(* Logix 5000 project; controller reports 1756-L63 rev 20.11; software revision 20.04; part 27 of 52 *)

        [1912].log_data[0].min := 1.0, [1912].log_data[0].max := 1.0, [1912].log_data[0].total := 300.0, [1912].log_data[0].time := 300.0, [1912].log_data[0].minminute := 40, [1912].log_data[0].maxminute := 40, [1912].log_data[0].valid := 1, [1912].log_data[1].valid := 1, [1912].log_data[2].valid := 1, [1912].log_data[3].valid := 1, [1912].log_data[4].valid := 1, [1912].log_data[5].valid := 1, [1912].log_data[6].valid := 1, [1912].log_data[7].valid := 1, [1912].log_data[8].valid := 1, [1912].log_data[9].valid := 1, [1912].log_data[10].valid := 1, [1912].log_data[11].valid := 1, [1912].log_data[12].valid := 1, [1912].log_data[13].valid := 1, [1912].log_data[14].valid := 1, [1912].log_data[15].valid := 1, [1912].log_data[16].valid := 1, [1912].log_data[17].valid := 1, [1912].log_data[18].valid := 1, [1912].log_data[19].valid := 1, [1912].time.Year := 2023, [1912].time.Month := 1, [1912].time.Day := 16, [1912].time.Hour := 7, [1912].time.Minute := 44, [1912].time.Second := 59, [1913].log_data[0].min := 1.0, [1913].log_data[0].max := 1.0, [1913].log_data[0].total := 300.0, [1913].log_data[0].time := 300.0, [1913].log_data[0].minminute := 45, [1913].log_data[0].maxminute := 45, [1913].log_data[0].valid := 1, [1913].log_data[1].valid := 1, [1913].log_data[2].valid := 1, [1913].log_data[3].valid := 1, [1913].log_data[4].valid := 1, [1913].log_data[5].valid := 1, [1913].log_data[6].valid := 1, [1913].log_data[7].valid := 1, [1913].log_data[8].valid := 1, [1913].log_data[9].valid := 1, [1913].log_data[10].valid := 1, [1913].log_data[11].valid := 1, [1913].log_data[12].valid := 1, [1913].log_data[13].valid := 1, [1913].log_data[14].valid := 1, [1913].log_data[15].valid := 1, [1913].log_data[16].valid := 1, [1913].log_data[17].valid := 1, [1913].log_data[18].valid := 1, [1913].log_data[19].valid := 1, [1913].time.Year := 2023, [1913].time.Month := 1,
        [1913].time.Day := 16, [1913].time.Hour := 7, [1913].time.Minute := 49, [1913].time.Second := 59, [1914].log_data[0].min := 1.0, [1914].log_data[0].max := 1.0, [1914].log_data[0].total := 300.0, [1914].log_data[0].time := 300.0, [1914].log_data[0].minminute := 50, [1914].log_data[0].maxminute := 50, [1914].log_data[0].valid := 1, [1914].log_data[1].valid := 1, [1914].log_data[2].valid := 1, [1914].log_data[3].valid := 1, [1914].log_data[4].valid := 1, [1914].log_data[5].valid := 1, [1914].log_data[6].valid := 1, [1914].log_data[7].valid := 1, [1914].log_data[8].valid := 1, [1914].log_data[9].valid := 1, [1914].log_data[10].valid := 1, [1914].log_data[11].valid := 1, [1914].log_data[12].valid := 1, [1914].log_data[13].valid := 1, [1914].log_data[14].valid := 1, [1914].log_data[15].valid := 1, [1914].log_data[16].valid := 1, [1914].log_data[17].valid := 1, [1914].log_data[18].valid := 1, [1914].log_data[19].valid := 1, [1914].time.Year := 2023, [1914].time.Month := 1, [1914].time.Day := 16, [1914].time.Hour := 7, [1914].time.Minute := 54, [1914].time.Second := 59, [1915].log_data[0].min := 1.0, [1915].log_data[0].max := 1.0, [1915].log_data[0].total := 300.0, [1915].log_data[0].time := 300.0, [1915].log_data[0].minminute := 55, [1915].log_data[0].maxminute := 55, [1915].log_data[0].valid := 1, [1915].log_data[1].valid := 1, [1915].log_data[2].valid := 1, [1915].log_data[3].valid := 1, [1915].log_data[4].valid := 1, [1915].log_data[5].valid := 1, [1915].log_data[6].valid := 1, [1915].log_data[7].valid := 1, [1915].log_data[8].valid := 1, [1915].log_data[9].valid := 1, [1915].log_data[10].valid := 1, [1915].log_data[11].valid := 1, [1915].log_data[12].valid := 1, [1915].log_data[13].valid := 1, [1915].log_data[14].valid := 1, [1915].log_data[15].valid := 1, [1915].log_data[16].valid := 1, [1915].log_data[17].valid := 1,
        [1915].log_data[18].valid := 1, [1915].log_data[19].valid := 1, [1915].time.Year := 2023, [1915].time.Month := 1, [1915].time.Day := 16, [1915].time.Hour := 7, [1915].time.Minute := 59, [1915].time.Second := 59, [1916].log_data[0].min := 1.0, [1916].log_data[0].max := 1.0, [1916].log_data[0].total := 300.0, [1916].log_data[0].time := 300.0, [1916].log_data[0].valid := 1, [1916].log_data[1].valid := 1, [1916].log_data[2].valid := 1, [1916].log_data[3].valid := 1, [1916].log_data[4].valid := 1, [1916].log_data[5].valid := 1, [1916].log_data[6].valid := 1, [1916].log_data[7].valid := 1, [1916].log_data[8].valid := 1, [1916].log_data[9].valid := 1, [1916].log_data[10].valid := 1, [1916].log_data[11].valid := 1, [1916].log_data[12].valid := 1, [1916].log_data[13].valid := 1, [1916].log_data[14].valid := 1, [1916].log_data[15].valid := 1, [1916].log_data[16].valid := 1, [1916].log_data[17].valid := 1, [1916].log_data[18].valid := 1, [1916].log_data[19].valid := 1, [1916].time.Year := 2023, [1916].time.Month := 1, [1916].time.Day := 16, [1916].time.Hour := 8, [1916].time.Minute := 4, [1916].time.Second := 59, [1917].log_data[0].min := 1.0, [1917].log_data[0].max := 1.0, [1917].log_data[0].total := 300.0, [1917].log_data[0].time := 300.0, [1917].log_data[0].minminute := 5, [1917].log_data[0].maxminute := 5, [1917].log_data[0].valid := 1, [1917].log_data[1].valid := 1, [1917].log_data[2].valid := 1, [1917].log_data[3].valid := 1, [1917].log_data[4].valid := 1, [1917].log_data[5].valid := 1, [1917].log_data[6].valid := 1, [1917].log_data[7].valid := 1, [1917].log_data[8].valid := 1, [1917].log_data[9].valid := 1, [1917].log_data[10].valid := 1, [1917].log_data[11].valid := 1, [1917].log_data[12].valid := 1, [1917].log_data[13].valid := 1, [1917].log_data[14].valid := 1, [1917].log_data[15].valid := 1,
        [1917].log_data[16].valid := 1, [1917].log_data[17].valid := 1, [1917].log_data[18].valid := 1, [1917].log_data[19].valid := 1, [1917].time.Year := 2023, [1917].time.Month := 1, [1917].time.Day := 16, [1917].time.Hour := 8, [1917].time.Minute := 9, [1917].time.Second := 59, [1918].log_data[0].min := 1.0, [1918].log_data[0].max := 1.0, [1918].log_data[0].total := 300.0, [1918].log_data[0].time := 300.0, [1918].log_data[0].minminute := 10, [1918].log_data[0].maxminute := 10, [1918].log_data[0].valid := 1, [1918].log_data[1].valid := 1, [1918].log_data[2].valid := 1, [1918].log_data[3].valid := 1, [1918].log_data[4].valid := 1, [1918].log_data[5].valid := 1, [1918].log_data[6].valid := 1, [1918].log_data[7].valid := 1, [1918].log_data[8].valid := 1, [1918].log_data[9].valid := 1, [1918].log_data[10].valid := 1, [1918].log_data[11].valid := 1, [1918].log_data[12].valid := 1, [1918].log_data[13].valid := 1, [1918].log_data[14].valid := 1, [1918].log_data[15].valid := 1, [1918].log_data[16].valid := 1, [1918].log_data[17].valid := 1, [1918].log_data[18].valid := 1, [1918].log_data[19].valid := 1, [1918].time.Year := 2023, [1918].time.Month := 1, [1918].time.Day := 16, [1918].time.Hour := 8, [1918].time.Minute := 14, [1918].time.Second := 59, [1919].log_data[0].min := 1.0, [1919].log_data[0].max := 1.0, [1919].log_data[0].total := 300.0, [1919].log_data[0].time := 300.0, [1919].log_data[0].minminute := 15, [1919].log_data[0].maxminute := 15, [1919].log_data[0].valid := 1, [1919].log_data[1].valid := 1, [1919].log_data[2].valid := 1, [1919].log_data[3].valid := 1, [1919].log_data[4].valid := 1, [1919].log_data[5].valid := 1, [1919].log_data[6].valid := 1, [1919].log_data[7].valid := 1, [1919].log_data[8].valid := 1, [1919].log_data[9].valid := 1, [1919].log_data[10].valid := 1, [1919].log_data[11].valid := 1,
        [1919].log_data[12].valid := 1, [1919].log_data[13].valid := 1, [1919].log_data[14].valid := 1, [1919].log_data[15].valid := 1, [1919].log_data[16].valid := 1, [1919].log_data[17].valid := 1, [1919].log_data[18].valid := 1, [1919].log_data[19].valid := 1, [1919].time.Year := 2023, [1919].time.Month := 1, [1919].time.Day := 16, [1919].time.Hour := 8, [1919].time.Minute := 19, [1919].time.Second := 59, [1920].log_data[0].min := 1.0, [1920].log_data[0].max := 1.0, [1920].log_data[0].total := 300.0, [1920].log_data[0].time := 300.0, [1920].log_data[0].minminute := 20, [1920].log_data[0].maxminute := 20, [1920].log_data[0].valid := 1, [1920].log_data[1].valid := 1, [1920].log_data[2].valid := 1, [1920].log_data[3].valid := 1, [1920].log_data[4].valid := 1, [1920].log_data[5].valid := 1, [1920].log_data[6].valid := 1, [1920].log_data[7].valid := 1, [1920].log_data[8].valid := 1, [1920].log_data[9].valid := 1, [1920].log_data[10].valid := 1, [1920].log_data[11].valid := 1, [1920].log_data[12].valid := 1, [1920].log_data[13].valid := 1, [1920].log_data[14].valid := 1, [1920].log_data[15].valid := 1, [1920].log_data[16].valid := 1, [1920].log_data[17].valid := 1, [1920].log_data[18].valid := 1, [1920].log_data[19].valid := 1, [1920].time.Year := 2023, [1920].time.Month := 1, [1920].time.Day := 16, [1920].time.Hour := 8, [1920].time.Minute := 24, [1920].time.Second := 59, [1921].log_data[0].min := 1.0, [1921].log_data[0].max := 1.0, [1921].log_data[0].total := 300.0, [1921].log_data[0].time := 300.0, [1921].log_data[0].minminute := 25, [1921].log_data[0].maxminute := 25, [1921].log_data[0].valid := 1, [1921].log_data[1].valid := 1, [1921].log_data[2].valid := 1, [1921].log_data[3].valid := 1, [1921].log_data[4].valid := 1, [1921].log_data[5].valid := 1, [1921].log_data[6].valid := 1, [1921].log_data[7].valid := 1,
        [1921].log_data[8].valid := 1, [1921].log_data[9].valid := 1, [1921].log_data[10].valid := 1, [1921].log_data[11].valid := 1, [1921].log_data[12].valid := 1, [1921].log_data[13].valid := 1, [1921].log_data[14].valid := 1, [1921].log_data[15].valid := 1, [1921].log_data[16].valid := 1, [1921].log_data[17].valid := 1, [1921].log_data[18].valid := 1, [1921].log_data[19].valid := 1, [1921].time.Year := 2023, [1921].time.Month := 1, [1921].time.Day := 16, [1921].time.Hour := 8, [1921].time.Minute := 29, [1921].time.Second := 59, [1922].log_data[0].min := 1.0, [1922].log_data[0].max := 1.0, [1922].log_data[0].total := 300.0, [1922].log_data[0].time := 300.0, [1922].log_data[0].minminute := 30, [1922].log_data[0].maxminute := 30, [1922].log_data[0].valid := 1, [1922].log_data[1].valid := 1, [1922].log_data[2].valid := 1, [1922].log_data[3].valid := 1, [1922].log_data[4].valid := 1, [1922].log_data[5].valid := 1, [1922].log_data[6].valid := 1, [1922].log_data[7].valid := 1, [1922].log_data[8].valid := 1, [1922].log_data[9].valid := 1, [1922].log_data[10].valid := 1, [1922].log_data[11].valid := 1, [1922].log_data[12].valid := 1, [1922].log_data[13].valid := 1, [1922].log_data[14].valid := 1, [1922].log_data[15].valid := 1, [1922].log_data[16].valid := 1, [1922].log_data[17].valid := 1, [1922].log_data[18].valid := 1, [1922].log_data[19].valid := 1, [1922].time.Year := 2023, [1922].time.Month := 1, [1922].time.Day := 16, [1922].time.Hour := 8, [1922].time.Minute := 34, [1922].time.Second := 59, [1923].log_data[0].min := 1.0, [1923].log_data[0].max := 1.0, [1923].log_data[0].total := 300.0, [1923].log_data[0].time := 300.0, [1923].log_data[0].minminute := 35, [1923].log_data[0].maxminute := 35, [1923].log_data[0].valid := 1, [1923].log_data[1].valid := 1, [1923].log_data[2].valid := 1, [1923].log_data[3].valid := 1,
        [1923].log_data[4].valid := 1, [1923].log_data[5].valid := 1, [1923].log_data[6].valid := 1, [1923].log_data[7].valid := 1, [1923].log_data[8].valid := 1, [1923].log_data[9].valid := 1, [1923].log_data[10].valid := 1, [1923].log_data[11].valid := 1, [1923].log_data[12].valid := 1, [1923].log_data[13].valid := 1, [1923].log_data[14].valid := 1, [1923].log_data[15].valid := 1, [1923].log_data[16].valid := 1, [1923].log_data[17].valid := 1, [1923].log_data[18].valid := 1, [1923].log_data[19].valid := 1, [1923].time.Year := 2023, [1923].time.Month := 1, [1923].time.Day := 16, [1923].time.Hour := 8, [1923].time.Minute := 39, [1923].time.Second := 59, [1924].log_data[0].min := 1.0, [1924].log_data[0].max := 1.0, [1924].log_data[0].total := 300.0, [1924].log_data[0].time := 300.0, [1924].log_data[0].minminute := 40, [1924].log_data[0].maxminute := 40, [1924].log_data[0].valid := 1, [1924].log_data[1].valid := 1, [1924].log_data[2].valid := 1, [1924].log_data[3].valid := 1, [1924].log_data[4].valid := 1, [1924].log_data[5].valid := 1, [1924].log_data[6].valid := 1, [1924].log_data[7].valid := 1, [1924].log_data[8].valid := 1, [1924].log_data[9].valid := 1, [1924].log_data[10].valid := 1, [1924].log_data[11].valid := 1, [1924].log_data[12].valid := 1, [1924].log_data[13].valid := 1, [1924].log_data[14].valid := 1, [1924].log_data[15].valid := 1, [1924].log_data[16].valid := 1, [1924].log_data[17].valid := 1, [1924].log_data[18].valid := 1, [1924].log_data[19].valid := 1, [1924].time.Year := 2023, [1924].time.Month := 1, [1924].time.Day := 16, [1924].time.Hour := 8, [1924].time.Minute := 44, [1924].time.Second := 59, [1925].log_data[0].min := 1.0, [1925].log_data[0].max := 1.0, [1925].log_data[0].total := 300.0, [1925].log_data[0].time := 300.0, [1925].log_data[0].minminute := 45, [1925].log_data[0].maxminute := 45,
        [1925].log_data[0].valid := 1, [1925].log_data[1].valid := 1, [1925].log_data[2].valid := 1, [1925].log_data[3].valid := 1, [1925].log_data[4].valid := 1, [1925].log_data[5].valid := 1, [1925].log_data[6].valid := 1, [1925].log_data[7].valid := 1, [1925].log_data[8].valid := 1, [1925].log_data[9].valid := 1, [1925].log_data[10].valid := 1, [1925].log_data[11].valid := 1, [1925].log_data[12].valid := 1, [1925].log_data[13].valid := 1, [1925].log_data[14].valid := 1, [1925].log_data[15].valid := 1, [1925].log_data[16].valid := 1, [1925].log_data[17].valid := 1, [1925].log_data[18].valid := 1, [1925].log_data[19].valid := 1, [1925].time.Year := 2023, [1925].time.Month := 1, [1925].time.Day := 16, [1925].time.Hour := 8, [1925].time.Minute := 49, [1925].time.Second := 59, [1926].log_data[0].min := 1.0, [1926].log_data[0].max := 1.0, [1926].log_data[0].total := 300.0, [1926].log_data[0].time := 300.0, [1926].log_data[0].minminute := 50, [1926].log_data[0].maxminute := 50, [1926].log_data[0].valid := 1, [1926].log_data[1].valid := 1, [1926].log_data[2].valid := 1, [1926].log_data[3].valid := 1, [1926].log_data[4].valid := 1, [1926].log_data[5].valid := 1, [1926].log_data[6].valid := 1, [1926].log_data[7].valid := 1, [1926].log_data[8].valid := 1, [1926].log_data[9].valid := 1, [1926].log_data[10].valid := 1, [1926].log_data[11].valid := 1, [1926].log_data[12].valid := 1, [1926].log_data[13].valid := 1, [1926].log_data[14].valid := 1, [1926].log_data[15].valid := 1, [1926].log_data[16].valid := 1, [1926].log_data[17].valid := 1, [1926].log_data[18].valid := 1, [1926].log_data[19].valid := 1, [1926].time.Year := 2023, [1926].time.Month := 1, [1926].time.Day := 16, [1926].time.Hour := 8, [1926].time.Minute := 54, [1926].time.Second := 59, [1927].log_data[0].min := 1.0, [1927].log_data[0].max := 1.0,
        [1927].log_data[0].total := 300.0, [1927].log_data[0].time := 300.0, [1927].log_data[0].minminute := 55, [1927].log_data[0].maxminute := 55, [1927].log_data[0].valid := 1, [1927].log_data[1].valid := 1, [1927].log_data[2].valid := 1, [1927].log_data[3].valid := 1, [1927].log_data[4].valid := 1, [1927].log_data[5].valid := 1, [1927].log_data[6].valid := 1, [1927].log_data[7].valid := 1, [1927].log_data[8].valid := 1, [1927].log_data[9].valid := 1, [1927].log_data[10].valid := 1, [1927].log_data[11].valid := 1, [1927].log_data[12].valid := 1, [1927].log_data[13].valid := 1, [1927].log_data[14].valid := 1, [1927].log_data[15].valid := 1, [1927].log_data[16].valid := 1, [1927].log_data[17].valid := 1, [1927].log_data[18].valid := 1, [1927].log_data[19].valid := 1, [1927].time.Year := 2023, [1927].time.Month := 1, [1927].time.Day := 16, [1927].time.Hour := 8, [1927].time.Minute := 59, [1927].time.Second := 59, [1928].log_data[0].min := 1.0, [1928].log_data[0].max := 1.0, [1928].log_data[0].total := 300.0, [1928].log_data[0].time := 300.0, [1928].log_data[0].valid := 1, [1928].log_data[1].valid := 1, [1928].log_data[2].valid := 1, [1928].log_data[3].valid := 1, [1928].log_data[4].valid := 1, [1928].log_data[5].valid := 1, [1928].log_data[6].valid := 1, [1928].log_data[7].valid := 1, [1928].log_data[8].valid := 1, [1928].log_data[9].valid := 1, [1928].log_data[10].valid := 1, [1928].log_data[11].valid := 1, [1928].log_data[12].valid := 1, [1928].log_data[13].valid := 1, [1928].log_data[14].valid := 1, [1928].log_data[15].valid := 1, [1928].log_data[16].valid := 1, [1928].log_data[17].valid := 1, [1928].log_data[18].valid := 1, [1928].log_data[19].valid := 1, [1928].time.Year := 2023, [1928].time.Month := 1, [1928].time.Day := 16, [1928].time.Hour := 9, [1928].time.Minute := 4, [1928].time.Second := 59,
        [1929].log_data[0].min := 1.0, [1929].log_data[0].max := 1.0, [1929].log_data[0].total := 300.0, [1929].log_data[0].time := 300.0, [1929].log_data[0].minminute := 5, [1929].log_data[0].maxminute := 5, [1929].log_data[0].valid := 1, [1929].log_data[1].valid := 1, [1929].log_data[2].valid := 1, [1929].log_data[3].valid := 1, [1929].log_data[4].valid := 1, [1929].log_data[5].valid := 1, [1929].log_data[6].valid := 1, [1929].log_data[7].valid := 1, [1929].log_data[8].valid := 1, [1929].log_data[9].valid := 1, [1929].log_data[10].valid := 1, [1929].log_data[11].valid := 1, [1929].log_data[12].valid := 1, [1929].log_data[13].valid := 1, [1929].log_data[14].valid := 1, [1929].log_data[15].valid := 1, [1929].log_data[16].valid := 1, [1929].log_data[17].valid := 1, [1929].log_data[18].valid := 1, [1929].log_data[19].valid := 1, [1929].time.Year := 2023, [1929].time.Month := 1, [1929].time.Day := 16, [1929].time.Hour := 9, [1929].time.Minute := 9, [1929].time.Second := 59, [1930].log_data[0].min := 1.0, [1930].log_data[0].max := 1.0, [1930].log_data[0].total := 300.0, [1930].log_data[0].time := 300.0, [1930].log_data[0].minminute := 10, [1930].log_data[0].maxminute := 10, [1930].log_data[0].valid := 1, [1930].log_data[1].valid := 1, [1930].log_data[2].valid := 1, [1930].log_data[3].valid := 1, [1930].log_data[4].valid := 1, [1930].log_data[5].valid := 1, [1930].log_data[6].valid := 1, [1930].log_data[7].valid := 1, [1930].log_data[8].valid := 1, [1930].log_data[9].valid := 1, [1930].log_data[10].valid := 1, [1930].log_data[11].valid := 1, [1930].log_data[12].valid := 1, [1930].log_data[13].valid := 1, [1930].log_data[14].valid := 1, [1930].log_data[15].valid := 1, [1930].log_data[16].valid := 1, [1930].log_data[17].valid := 1, [1930].log_data[18].valid := 1, [1930].log_data[19].valid := 1, [1930].time.Year := 2023, [1930].time.Month := 1,
        [1930].time.Day := 16, [1930].time.Hour := 9, [1930].time.Minute := 14, [1930].time.Second := 59, [1931].log_data[0].min := 1.0, [1931].log_data[0].max := 1.0, [1931].log_data[0].total := 300.0, [1931].log_data[0].time := 300.0, [1931].log_data[0].minminute := 15, [1931].log_data[0].maxminute := 15, [1931].log_data[0].valid := 1, [1931].log_data[1].valid := 1, [1931].log_data[2].valid := 1, [1931].log_data[3].valid := 1, [1931].log_data[4].valid := 1, [1931].log_data[5].valid := 1, [1931].log_data[6].valid := 1, [1931].log_data[7].valid := 1, [1931].log_data[8].valid := 1, [1931].log_data[9].valid := 1, [1931].log_data[10].valid := 1, [1931].log_data[11].valid := 1, [1931].log_data[12].valid := 1, [1931].log_data[13].valid := 1, [1931].log_data[14].valid := 1, [1931].log_data[15].valid := 1, [1931].log_data[16].valid := 1, [1931].log_data[17].valid := 1, [1931].log_data[18].valid := 1, [1931].log_data[19].valid := 1, [1931].time.Year := 2023, [1931].time.Month := 1, [1931].time.Day := 16, [1931].time.Hour := 9, [1931].time.Minute := 19, [1931].time.Second := 59, [1932].log_data[0].min := 1.0, [1932].log_data[0].max := 1.0, [1932].log_data[0].total := 300.0, [1932].log_data[0].time := 300.0, [1932].log_data[0].minminute := 20, [1932].log_data[0].maxminute := 20, [1932].log_data[0].valid := 1, [1932].log_data[1].valid := 1, [1932].log_data[2].valid := 1, [1932].log_data[3].valid := 1, [1932].log_data[4].valid := 1, [1932].log_data[5].valid := 1, [1932].log_data[6].valid := 1, [1932].log_data[7].valid := 1, [1932].log_data[8].valid := 1, [1932].log_data[9].valid := 1, [1932].log_data[10].valid := 1, [1932].log_data[11].valid := 1, [1932].log_data[12].valid := 1, [1932].log_data[13].valid := 1, [1932].log_data[14].valid := 1, [1932].log_data[15].valid := 1, [1932].log_data[16].valid := 1, [1932].log_data[17].valid := 1,
        [1932].log_data[18].valid := 1, [1932].log_data[19].valid := 1, [1932].time.Year := 2023, [1932].time.Month := 1, [1932].time.Day := 16, [1932].time.Hour := 9, [1932].time.Minute := 24, [1932].time.Second := 59, [1933].log_data[0].min := 1.0, [1933].log_data[0].max := 1.0, [1933].log_data[0].total := 300.0, [1933].log_data[0].time := 300.0, [1933].log_data[0].minminute := 25, [1933].log_data[0].maxminute := 25, [1933].log_data[0].valid := 1, [1933].log_data[1].valid := 1, [1933].log_data[2].valid := 1, [1933].log_data[3].valid := 1, [1933].log_data[4].valid := 1, [1933].log_data[5].valid := 1, [1933].log_data[6].valid := 1, [1933].log_data[7].valid := 1, [1933].log_data[8].valid := 1, [1933].log_data[9].valid := 1, [1933].log_data[10].valid := 1, [1933].log_data[11].valid := 1, [1933].log_data[12].valid := 1, [1933].log_data[13].valid := 1, [1933].log_data[14].valid := 1, [1933].log_data[15].valid := 1, [1933].log_data[16].valid := 1, [1933].log_data[17].valid := 1, [1933].log_data[18].valid := 1, [1933].log_data[19].valid := 1, [1933].time.Year := 2023, [1933].time.Month := 1, [1933].time.Day := 16, [1933].time.Hour := 9, [1933].time.Minute := 29, [1933].time.Second := 59, [1934].log_data[0].min := 1.0, [1934].log_data[0].max := 1.0, [1934].log_data[0].total := 300.0, [1934].log_data[0].time := 300.0, [1934].log_data[0].minminute := 30, [1934].log_data[0].maxminute := 30, [1934].log_data[0].valid := 1, [1934].log_data[1].valid := 1, [1934].log_data[2].valid := 1, [1934].log_data[3].valid := 1, [1934].log_data[4].valid := 1, [1934].log_data[5].valid := 1, [1934].log_data[6].valid := 1, [1934].log_data[7].valid := 1, [1934].log_data[8].valid := 1, [1934].log_data[9].valid := 1, [1934].log_data[10].valid := 1, [1934].log_data[11].valid := 1, [1934].log_data[12].valid := 1, [1934].log_data[13].valid := 1,
        [1934].log_data[14].valid := 1, [1934].log_data[15].valid := 1, [1934].log_data[16].valid := 1, [1934].log_data[17].valid := 1, [1934].log_data[18].valid := 1, [1934].log_data[19].valid := 1, [1934].time.Year := 2023, [1934].time.Month := 1, [1934].time.Day := 16, [1934].time.Hour := 9, [1934].time.Minute := 34, [1934].time.Second := 59, [1935].log_data[0].min := 1.0, [1935].log_data[0].max := 1.0, [1935].log_data[0].total := 300.0, [1935].log_data[0].time := 300.0, [1935].log_data[0].minminute := 35, [1935].log_data[0].maxminute := 35, [1935].log_data[0].valid := 1, [1935].log_data[1].valid := 1, [1935].log_data[2].valid := 1, [1935].log_data[3].valid := 1, [1935].log_data[4].valid := 1, [1935].log_data[5].valid := 1, [1935].log_data[6].valid := 1, [1935].log_data[7].valid := 1, [1935].log_data[8].valid := 1, [1935].log_data[9].valid := 1, [1935].log_data[10].valid := 1, [1935].log_data[11].valid := 1, [1935].log_data[12].valid := 1, [1935].log_data[13].valid := 1, [1935].log_data[14].valid := 1, [1935].log_data[15].valid := 1, [1935].log_data[16].valid := 1, [1935].log_data[17].valid := 1, [1935].log_data[18].valid := 1, [1935].log_data[19].valid := 1, [1935].time.Year := 2023, [1935].time.Month := 1, [1935].time.Day := 16, [1935].time.Hour := 9, [1935].time.Minute := 39, [1935].time.Second := 59, [1936].log_data[0].min := 1.0, [1936].log_data[0].max := 1.0, [1936].log_data[0].total := 300.0, [1936].log_data[0].time := 300.0, [1936].log_data[0].minminute := 40, [1936].log_data[0].maxminute := 40, [1936].log_data[0].valid := 1, [1936].log_data[1].valid := 1, [1936].log_data[2].valid := 1, [1936].log_data[3].valid := 1, [1936].log_data[4].valid := 1, [1936].log_data[5].valid := 1, [1936].log_data[6].valid := 1, [1936].log_data[7].valid := 1, [1936].log_data[8].valid := 1, [1936].log_data[9].valid := 1,
        [1936].log_data[10].valid := 1, [1936].log_data[11].valid := 1, [1936].log_data[12].valid := 1, [1936].log_data[13].valid := 1, [1936].log_data[14].valid := 1, [1936].log_data[15].valid := 1, [1936].log_data[16].valid := 1, [1936].log_data[17].valid := 1, [1936].log_data[18].valid := 1, [1936].log_data[19].valid := 1, [1936].time.Year := 2023, [1936].time.Month := 1, [1936].time.Day := 16, [1936].time.Hour := 9, [1936].time.Minute := 44, [1936].time.Second := 59, [1937].log_data[0].min := 1.0, [1937].log_data[0].max := 1.0, [1937].log_data[0].total := 300.0, [1937].log_data[0].time := 300.0, [1937].log_data[0].minminute := 45, [1937].log_data[0].maxminute := 45, [1937].log_data[0].valid := 1, [1937].log_data[1].valid := 1, [1937].log_data[2].valid := 1, [1937].log_data[3].valid := 1, [1937].log_data[4].valid := 1, [1937].log_data[5].valid := 1, [1937].log_data[6].valid := 1, [1937].log_data[7].valid := 1, [1937].log_data[8].valid := 1, [1937].log_data[9].valid := 1, [1937].log_data[10].valid := 1, [1937].log_data[11].valid := 1, [1937].log_data[12].valid := 1, [1937].log_data[13].valid := 1, [1937].log_data[14].valid := 1, [1937].log_data[15].valid := 1, [1937].log_data[16].valid := 1, [1937].log_data[17].valid := 1, [1937].log_data[18].valid := 1, [1937].log_data[19].valid := 1, [1937].time.Year := 2023, [1937].time.Month := 1, [1937].time.Day := 16, [1937].time.Hour := 9, [1937].time.Minute := 49, [1937].time.Second := 59, [1938].log_data[0].min := 1.0, [1938].log_data[0].max := 1.0, [1938].log_data[0].total := 300.0, [1938].log_data[0].time := 300.0, [1938].log_data[0].minminute := 50, [1938].log_data[0].maxminute := 50, [1938].log_data[0].valid := 1, [1938].log_data[1].valid := 1, [1938].log_data[2].valid := 1, [1938].log_data[3].valid := 1, [1938].log_data[4].valid := 1, [1938].log_data[5].valid := 1,
        [1938].log_data[6].valid := 1, [1938].log_data[7].valid := 1, [1938].log_data[8].valid := 1, [1938].log_data[9].valid := 1, [1938].log_data[10].valid := 1, [1938].log_data[11].valid := 1, [1938].log_data[12].valid := 1, [1938].log_data[13].valid := 1, [1938].log_data[14].valid := 1, [1938].log_data[15].valid := 1, [1938].log_data[16].valid := 1, [1938].log_data[17].valid := 1, [1938].log_data[18].valid := 1, [1938].log_data[19].valid := 1, [1938].time.Year := 2023, [1938].time.Month := 1, [1938].time.Day := 16, [1938].time.Hour := 9, [1938].time.Minute := 54, [1938].time.Second := 59, [1939].log_data[0].min := 1.0, [1939].log_data[0].max := 1.0, [1939].log_data[0].total := 300.0, [1939].log_data[0].time := 300.0, [1939].log_data[0].minminute := 55, [1939].log_data[0].maxminute := 55, [1939].log_data[0].valid := 1, [1939].log_data[1].valid := 1, [1939].log_data[2].valid := 1, [1939].log_data[3].valid := 1, [1939].log_data[4].valid := 1, [1939].log_data[5].valid := 1, [1939].log_data[6].valid := 1, [1939].log_data[7].valid := 1, [1939].log_data[8].valid := 1, [1939].log_data[9].valid := 1, [1939].log_data[10].valid := 1, [1939].log_data[11].valid := 1, [1939].log_data[12].valid := 1, [1939].log_data[13].valid := 1, [1939].log_data[14].valid := 1, [1939].log_data[15].valid := 1, [1939].log_data[16].valid := 1, [1939].log_data[17].valid := 1, [1939].log_data[18].valid := 1, [1939].log_data[19].valid := 1, [1939].time.Year := 2023, [1939].time.Month := 1, [1939].time.Day := 16, [1939].time.Hour := 9, [1939].time.Minute := 59, [1939].time.Second := 59, [1940].log_data[0].min := 1.0, [1940].log_data[0].max := 1.0, [1940].log_data[0].total := 299.5, [1940].log_data[0].time := 299.5, [1940].log_data[0].valid := 1, [1940].log_data[1].valid := 1, [1940].log_data[2].valid := 1, [1940].log_data[3].valid := 1,
        [1940].log_data[4].valid := 1, [1940].log_data[5].valid := 1, [1940].log_data[6].valid := 1, [1940].log_data[7].valid := 1, [1940].log_data[8].valid := 1, [1940].log_data[9].valid := 1, [1940].log_data[10].valid := 1, [1940].log_data[11].valid := 1, [1940].log_data[12].valid := 1, [1940].log_data[13].valid := 1, [1940].log_data[14].valid := 1, [1940].log_data[15].valid := 1, [1940].log_data[16].valid := 1, [1940].log_data[17].valid := 1, [1940].log_data[18].valid := 1, [1940].log_data[19].valid := 1, [1940].time.Year := 2023, [1940].time.Month := 1, [1940].time.Day := 16, [1940].time.Hour := 10, [1940].time.Minute := 4, [1940].time.Second := 59, [1941].log_data[0].min := 1.0, [1941].log_data[0].max := 1.0, [1941].log_data[0].total := 300.0, [1941].log_data[0].time := 300.0, [1941].log_data[0].minminute := 5, [1941].log_data[0].maxminute := 5, [1941].log_data[0].valid := 1, [1941].log_data[1].valid := 1, [1941].log_data[2].valid := 1, [1941].log_data[3].valid := 1, [1941].log_data[4].valid := 1, [1941].log_data[5].valid := 1, [1941].log_data[6].valid := 1, [1941].log_data[7].valid := 1, [1941].log_data[8].valid := 1, [1941].log_data[9].valid := 1, [1941].log_data[10].valid := 1, [1941].log_data[11].valid := 1, [1941].log_data[12].valid := 1, [1941].log_data[13].valid := 1, [1941].log_data[14].valid := 1, [1941].log_data[15].valid := 1, [1941].log_data[16].valid := 1, [1941].log_data[17].valid := 1, [1941].log_data[18].valid := 1, [1941].log_data[19].valid := 1, [1941].time.Year := 2023, [1941].time.Month := 1, [1941].time.Day := 16, [1941].time.Hour := 10, [1941].time.Minute := 9, [1941].time.Second := 59, [1942].log_data[0].min := 1.0, [1942].log_data[0].max := 1.0, [1942].log_data[0].total := 300.0, [1942].log_data[0].time := 300.0, [1942].log_data[0].minminute := 10, [1942].log_data[0].maxminute := 10,
        [1942].log_data[0].valid := 1, [1942].log_data[1].valid := 1, [1942].log_data[2].valid := 1, [1942].log_data[3].valid := 1, [1942].log_data[4].valid := 1, [1942].log_data[5].valid := 1, [1942].log_data[6].valid := 1, [1942].log_data[7].valid := 1, [1942].log_data[8].valid := 1, [1942].log_data[9].valid := 1, [1942].log_data[10].valid := 1, [1942].log_data[11].valid := 1, [1942].log_data[12].valid := 1, [1942].log_data[13].valid := 1, [1942].log_data[14].valid := 1, [1942].log_data[15].valid := 1, [1942].log_data[16].valid := 1, [1942].log_data[17].valid := 1, [1942].log_data[18].valid := 1, [1942].log_data[19].valid := 1, [1942].time.Year := 2023, [1942].time.Month := 1, [1942].time.Day := 16, [1942].time.Hour := 10, [1942].time.Minute := 14, [1942].time.Second := 59, [1943].log_data[0].min := 1.0, [1943].log_data[0].max := 1.0, [1943].log_data[0].total := 300.0, [1943].log_data[0].time := 300.0, [1943].log_data[0].minminute := 15, [1943].log_data[0].maxminute := 15, [1943].log_data[0].valid := 1, [1943].log_data[1].valid := 1, [1943].log_data[2].valid := 1, [1943].log_data[3].valid := 1, [1943].log_data[4].valid := 1, [1943].log_data[5].valid := 1, [1943].log_data[6].valid := 1, [1943].log_data[7].valid := 1, [1943].log_data[8].valid := 1, [1943].log_data[9].valid := 1, [1943].log_data[10].valid := 1, [1943].log_data[11].valid := 1, [1943].log_data[12].valid := 1, [1943].log_data[13].valid := 1, [1943].log_data[14].valid := 1, [1943].log_data[15].valid := 1, [1943].log_data[16].valid := 1, [1943].log_data[17].valid := 1, [1943].log_data[18].valid := 1, [1943].log_data[19].valid := 1, [1943].time.Year := 2023, [1943].time.Month := 1, [1943].time.Day := 16, [1943].time.Hour := 10, [1943].time.Minute := 19, [1943].time.Second := 59, [1944].log_data[0].min := 1.0, [1944].log_data[0].max := 1.0,
        [1944].log_data[0].total := 300.0, [1944].log_data[0].time := 300.0, [1944].log_data[0].minminute := 20, [1944].log_data[0].maxminute := 20, [1944].log_data[0].valid := 1, [1944].log_data[1].valid := 1, [1944].log_data[2].valid := 1, [1944].log_data[3].valid := 1, [1944].log_data[4].valid := 1, [1944].log_data[5].valid := 1, [1944].log_data[6].valid := 1, [1944].log_data[7].valid := 1, [1944].log_data[8].valid := 1, [1944].log_data[9].valid := 1, [1944].log_data[10].valid := 1, [1944].log_data[11].valid := 1, [1944].log_data[12].valid := 1, [1944].log_data[13].valid := 1, [1944].log_data[14].valid := 1, [1944].log_data[15].valid := 1, [1944].log_data[16].valid := 1, [1944].log_data[17].valid := 1, [1944].log_data[18].valid := 1, [1944].log_data[19].valid := 1, [1944].time.Year := 2023, [1944].time.Month := 1, [1944].time.Day := 16, [1944].time.Hour := 10, [1944].time.Minute := 24, [1944].time.Second := 59, [1945].log_data[0].min := 1.0, [1945].log_data[0].max := 1.0, [1945].log_data[0].total := 300.0, [1945].log_data[0].time := 300.0, [1945].log_data[0].minminute := 25, [1945].log_data[0].maxminute := 25, [1945].log_data[0].valid := 1, [1945].log_data[1].valid := 1, [1945].log_data[2].valid := 1, [1945].log_data[3].valid := 1, [1945].log_data[4].valid := 1, [1945].log_data[5].valid := 1, [1945].log_data[6].valid := 1, [1945].log_data[7].valid := 1, [1945].log_data[8].valid := 1, [1945].log_data[9].valid := 1, [1945].log_data[10].valid := 1, [1945].log_data[11].valid := 1, [1945].log_data[12].valid := 1, [1945].log_data[13].valid := 1, [1945].log_data[14].valid := 1, [1945].log_data[15].valid := 1, [1945].log_data[16].valid := 1, [1945].log_data[17].valid := 1, [1945].log_data[18].valid := 1, [1945].log_data[19].valid := 1, [1945].time.Year := 2023, [1945].time.Month := 1, [1945].time.Day := 16, [1945].time.Hour := 10,
        [1945].time.Minute := 29, [1945].time.Second := 59, [1946].log_data[0].min := 1.0, [1946].log_data[0].max := 1.0, [1946].log_data[0].total := 300.0, [1946].log_data[0].time := 300.0, [1946].log_data[0].minminute := 30, [1946].log_data[0].maxminute := 30, [1946].log_data[0].valid := 1, [1946].log_data[1].valid := 1, [1946].log_data[2].valid := 1, [1946].log_data[3].valid := 1, [1946].log_data[4].valid := 1, [1946].log_data[5].valid := 1, [1946].log_data[6].valid := 1, [1946].log_data[7].valid := 1, [1946].log_data[8].valid := 1, [1946].log_data[9].valid := 1, [1946].log_data[10].valid := 1, [1946].log_data[11].valid := 1, [1946].log_data[12].valid := 1, [1946].log_data[13].valid := 1, [1946].log_data[14].valid := 1, [1946].log_data[15].valid := 1, [1946].log_data[16].valid := 1, [1946].log_data[17].valid := 1, [1946].log_data[18].valid := 1, [1946].log_data[19].valid := 1, [1946].time.Year := 2023, [1946].time.Month := 1, [1946].time.Day := 16, [1946].time.Hour := 10, [1946].time.Minute := 34, [1946].time.Second := 59, [1947].log_data[0].min := 1.0, [1947].log_data[0].max := 1.0, [1947].log_data[0].total := 300.0, [1947].log_data[0].time := 300.0, [1947].log_data[0].minminute := 35, [1947].log_data[0].maxminute := 35, [1947].log_data[0].valid := 1, [1947].log_data[1].valid := 1, [1947].log_data[2].valid := 1, [1947].log_data[3].valid := 1, [1947].log_data[4].valid := 1, [1947].log_data[5].valid := 1, [1947].log_data[6].valid := 1, [1947].log_data[7].valid := 1, [1947].log_data[8].valid := 1, [1947].log_data[9].valid := 1, [1947].log_data[10].valid := 1, [1947].log_data[11].valid := 1, [1947].log_data[12].valid := 1, [1947].log_data[13].valid := 1, [1947].log_data[14].valid := 1, [1947].log_data[15].valid := 1, [1947].log_data[16].valid := 1, [1947].log_data[17].valid := 1, [1947].log_data[18].valid := 1, [1947].log_data[19].valid := 1,
        [1947].time.Year := 2023, [1947].time.Month := 1, [1947].time.Day := 16, [1947].time.Hour := 10, [1947].time.Minute := 39, [1947].time.Second := 59, [1948].log_data[0].min := 1.0, [1948].log_data[0].max := 1.0, [1948].log_data[0].total := 300.0, [1948].log_data[0].time := 300.0, [1948].log_data[0].minminute := 40, [1948].log_data[0].maxminute := 40, [1948].log_data[0].valid := 1, [1948].log_data[1].valid := 1, [1948].log_data[2].valid := 1, [1948].log_data[3].valid := 1, [1948].log_data[4].valid := 1, [1948].log_data[5].valid := 1, [1948].log_data[6].valid := 1, [1948].log_data[7].valid := 1, [1948].log_data[8].valid := 1, [1948].log_data[9].valid := 1, [1948].log_data[10].valid := 1, [1948].log_data[11].valid := 1, [1948].log_data[12].valid := 1, [1948].log_data[13].valid := 1, [1948].log_data[14].valid := 1, [1948].log_data[15].valid := 1, [1948].log_data[16].valid := 1, [1948].log_data[17].valid := 1, [1948].log_data[18].valid := 1, [1948].log_data[19].valid := 1, [1948].time.Year := 2023, [1948].time.Month := 1, [1948].time.Day := 16, [1948].time.Hour := 10, [1948].time.Minute := 44, [1948].time.Second := 59, [1949].log_data[0].min := 1.0, [1949].log_data[0].max := 1.0, [1949].log_data[0].total := 300.0, [1949].log_data[0].time := 300.0, [1949].log_data[0].minminute := 45, [1949].log_data[0].maxminute := 45, [1949].log_data[0].valid := 1, [1949].log_data[1].valid := 1, [1949].log_data[2].valid := 1, [1949].log_data[3].valid := 1, [1949].log_data[4].valid := 1, [1949].log_data[5].valid := 1, [1949].log_data[6].valid := 1, [1949].log_data[7].valid := 1, [1949].log_data[8].valid := 1, [1949].log_data[9].valid := 1, [1949].log_data[10].valid := 1, [1949].log_data[11].valid := 1, [1949].log_data[12].valid := 1, [1949].log_data[13].valid := 1, [1949].log_data[14].valid := 1, [1949].log_data[15].valid := 1,
        [1949].log_data[16].valid := 1, [1949].log_data[17].valid := 1, [1949].log_data[18].valid := 1, [1949].log_data[19].valid := 1, [1949].time.Year := 2023, [1949].time.Month := 1, [1949].time.Day := 16, [1949].time.Hour := 10, [1949].time.Minute := 49, [1949].time.Second := 59, [1950].log_data[0].min := 1.0, [1950].log_data[0].max := 1.0, [1950].log_data[0].total := 300.0, [1950].log_data[0].time := 300.0, [1950].log_data[0].minminute := 50, [1950].log_data[0].maxminute := 50, [1950].log_data[0].valid := 1, [1950].log_data[1].valid := 1, [1950].log_data[2].valid := 1, [1950].log_data[3].valid := 1, [1950].log_data[4].valid := 1, [1950].log_data[5].valid := 1, [1950].log_data[6].valid := 1, [1950].log_data[7].valid := 1, [1950].log_data[8].valid := 1, [1950].log_data[9].valid := 1, [1950].log_data[10].valid := 1, [1950].log_data[11].valid := 1, [1950].log_data[12].valid := 1, [1950].log_data[13].valid := 1, [1950].log_data[14].valid := 1, [1950].log_data[15].valid := 1, [1950].log_data[16].valid := 1, [1950].log_data[17].valid := 1, [1950].log_data[18].valid := 1, [1950].log_data[19].valid := 1, [1950].time.Year := 2023, [1950].time.Month := 1, [1950].time.Day := 16, [1950].time.Hour := 10, [1950].time.Minute := 54, [1950].time.Second := 59, [1951].log_data[0].min := 1.0, [1951].log_data[0].max := 1.0, [1951].log_data[0].total := 300.0, [1951].log_data[0].time := 300.0, [1951].log_data[0].minminute := 55, [1951].log_data[0].maxminute := 55, [1951].log_data[0].valid := 1, [1951].log_data[1].valid := 1, [1951].log_data[2].valid := 1, [1951].log_data[3].valid := 1, [1951].log_data[4].valid := 1, [1951].log_data[5].valid := 1, [1951].log_data[6].valid := 1, [1951].log_data[7].valid := 1, [1951].log_data[8].valid := 1, [1951].log_data[9].valid := 1, [1951].log_data[10].valid := 1, [1951].log_data[11].valid := 1,
        [1951].log_data[12].valid := 1, [1951].log_data[13].valid := 1, [1951].log_data[14].valid := 1, [1951].log_data[15].valid := 1, [1951].log_data[16].valid := 1, [1951].log_data[17].valid := 1, [1951].log_data[18].valid := 1, [1951].log_data[19].valid := 1, [1951].time.Year := 2023, [1951].time.Month := 1, [1951].time.Day := 16, [1951].time.Hour := 10, [1951].time.Minute := 59, [1951].time.Second := 59, [1952].log_data[0].min := 1.0, [1952].log_data[0].max := 1.0, [1952].log_data[0].total := 300.0, [1952].log_data[0].time := 300.0, [1952].log_data[0].valid := 1, [1952].log_data[1].valid := 1, [1952].log_data[2].valid := 1, [1952].log_data[3].valid := 1, [1952].log_data[4].valid := 1, [1952].log_data[5].valid := 1, [1952].log_data[6].valid := 1, [1952].log_data[7].valid := 1, [1952].log_data[8].valid := 1, [1952].log_data[9].valid := 1, [1952].log_data[10].valid := 1, [1952].log_data[11].valid := 1, [1952].log_data[12].valid := 1, [1952].log_data[13].valid := 1, [1952].log_data[14].valid := 1, [1952].log_data[15].valid := 1, [1952].log_data[16].valid := 1, [1952].log_data[17].valid := 1, [1952].log_data[18].valid := 1, [1952].log_data[19].valid := 1, [1952].time.Year := 2023, [1952].time.Month := 1, [1952].time.Day := 16, [1952].time.Hour := 11, [1952].time.Minute := 4, [1952].time.Second := 59, [1953].log_data[0].min := 1.0, [1953].log_data[0].max := 1.0, [1953].log_data[0].total := 300.0, [1953].log_data[0].time := 300.0, [1953].log_data[0].minminute := 5, [1953].log_data[0].maxminute := 5, [1953].log_data[0].valid := 1, [1953].log_data[1].valid := 1, [1953].log_data[2].valid := 1, [1953].log_data[3].valid := 1, [1953].log_data[4].valid := 1, [1953].log_data[5].valid := 1, [1953].log_data[6].valid := 1, [1953].log_data[7].valid := 1, [1953].log_data[8].valid := 1, [1953].log_data[9].valid := 1,
        [1953].log_data[10].valid := 1, [1953].log_data[11].valid := 1, [1953].log_data[12].valid := 1, [1953].log_data[13].valid := 1, [1953].log_data[14].valid := 1, [1953].log_data[15].valid := 1, [1953].log_data[16].valid := 1, [1953].log_data[17].valid := 1, [1953].log_data[18].valid := 1, [1953].log_data[19].valid := 1, [1953].time.Year := 2023, [1953].time.Month := 1, [1953].time.Day := 16, [1953].time.Hour := 11, [1953].time.Minute := 9, [1953].time.Second := 59, [1954].log_data[0].min := 1.0, [1954].log_data[0].max := 1.0, [1954].log_data[0].total := 300.0, [1954].log_data[0].time := 300.0, [1954].log_data[0].minminute := 10, [1954].log_data[0].maxminute := 10, [1954].log_data[0].valid := 1, [1954].log_data[1].valid := 1, [1954].log_data[2].valid := 1, [1954].log_data[3].valid := 1, [1954].log_data[4].valid := 1, [1954].log_data[5].valid := 1, [1954].log_data[6].valid := 1, [1954].log_data[7].valid := 1, [1954].log_data[8].valid := 1, [1954].log_data[9].valid := 1, [1954].log_data[10].valid := 1, [1954].log_data[11].valid := 1, [1954].log_data[12].valid := 1, [1954].log_data[13].valid := 1, [1954].log_data[14].valid := 1, [1954].log_data[15].valid := 1, [1954].log_data[16].valid := 1, [1954].log_data[17].valid := 1, [1954].log_data[18].valid := 1, [1954].log_data[19].valid := 1, [1954].time.Year := 2023, [1954].time.Month := 1, [1954].time.Day := 16, [1954].time.Hour := 11, [1954].time.Minute := 14, [1954].time.Second := 59, [1955].log_data[0].min := 1.0, [1955].log_data[0].max := 1.0, [1955].log_data[0].total := 300.0, [1955].log_data[0].time := 300.0, [1955].log_data[0].minminute := 15, [1955].log_data[0].maxminute := 15, [1955].log_data[0].valid := 1, [1955].log_data[1].valid := 1, [1955].log_data[2].valid := 1, [1955].log_data[3].valid := 1, [1955].log_data[4].valid := 1, [1955].log_data[5].valid := 1,
        [1955].log_data[6].valid := 1, [1955].log_data[7].valid := 1, [1955].log_data[8].valid := 1, [1955].log_data[9].valid := 1, [1955].log_data[10].valid := 1, [1955].log_data[11].valid := 1, [1955].log_data[12].valid := 1, [1955].log_data[13].valid := 1, [1955].log_data[14].valid := 1, [1955].log_data[15].valid := 1, [1955].log_data[16].valid := 1, [1955].log_data[17].valid := 1, [1955].log_data[18].valid := 1, [1955].log_data[19].valid := 1, [1955].time.Year := 2023, [1955].time.Month := 1, [1955].time.Day := 16, [1955].time.Hour := 11, [1955].time.Minute := 19, [1955].time.Second := 59, [1956].log_data[0].min := 1.0, [1956].log_data[0].max := 1.0, [1956].log_data[0].total := 300.0, [1956].log_data[0].time := 300.0, [1956].log_data[0].minminute := 20, [1956].log_data[0].maxminute := 20, [1956].log_data[0].valid := 1, [1956].log_data[1].valid := 1, [1956].log_data[2].valid := 1, [1956].log_data[3].valid := 1, [1956].log_data[4].valid := 1, [1956].log_data[5].valid := 1, [1956].log_data[6].valid := 1, [1956].log_data[7].valid := 1, [1956].log_data[8].valid := 1, [1956].log_data[9].valid := 1, [1956].log_data[10].valid := 1, [1956].log_data[11].valid := 1, [1956].log_data[12].valid := 1, [1956].log_data[13].valid := 1, [1956].log_data[14].valid := 1, [1956].log_data[15].valid := 1, [1956].log_data[16].valid := 1, [1956].log_data[17].valid := 1, [1956].log_data[18].valid := 1, [1956].log_data[19].valid := 1, [1956].time.Year := 2023, [1956].time.Month := 1, [1956].time.Day := 16, [1956].time.Hour := 11, [1956].time.Minute := 24, [1956].time.Second := 59, [1957].log_data[0].min := 1.0, [1957].log_data[0].max := 1.0, [1957].log_data[0].total := 300.0, [1957].log_data[0].time := 300.0, [1957].log_data[0].minminute := 25, [1957].log_data[0].maxminute := 25, [1957].log_data[0].valid := 1, [1957].log_data[1].valid := 1,
        [1957].log_data[2].valid := 1, [1957].log_data[3].valid := 1, [1957].log_data[4].valid := 1, [1957].log_data[5].valid := 1, [1957].log_data[6].valid := 1, [1957].log_data[7].valid := 1, [1957].log_data[8].valid := 1, [1957].log_data[9].valid := 1, [1957].log_data[10].valid := 1, [1957].log_data[11].valid := 1, [1957].log_data[12].valid := 1, [1957].log_data[13].valid := 1, [1957].log_data[14].valid := 1, [1957].log_data[15].valid := 1, [1957].log_data[16].valid := 1, [1957].log_data[17].valid := 1, [1957].log_data[18].valid := 1, [1957].log_data[19].valid := 1, [1957].time.Year := 2023, [1957].time.Month := 1, [1957].time.Day := 16, [1957].time.Hour := 11, [1957].time.Minute := 29, [1957].time.Second := 59, [1958].log_data[0].min := 1.0, [1958].log_data[0].max := 1.0, [1958].log_data[0].total := 300.0, [1958].log_data[0].time := 300.0, [1958].log_data[0].minminute := 30, [1958].log_data[0].maxminute := 30, [1958].log_data[0].valid := 1, [1958].log_data[1].valid := 1, [1958].log_data[2].valid := 1, [1958].log_data[3].valid := 1, [1958].log_data[4].valid := 1, [1958].log_data[5].valid := 1, [1958].log_data[6].valid := 1, [1958].log_data[7].valid := 1, [1958].log_data[8].valid := 1, [1958].log_data[9].valid := 1, [1958].log_data[10].valid := 1, [1958].log_data[11].valid := 1, [1958].log_data[12].valid := 1, [1958].log_data[13].valid := 1, [1958].log_data[14].valid := 1, [1958].log_data[15].valid := 1, [1958].log_data[16].valid := 1, [1958].log_data[17].valid := 1, [1958].log_data[18].valid := 1, [1958].log_data[19].valid := 1, [1958].time.Year := 2023, [1958].time.Month := 1, [1958].time.Day := 16, [1958].time.Hour := 11, [1958].time.Minute := 34, [1958].time.Second := 59, [1959].log_data[0].min := 1.0, [1959].log_data[0].max := 1.0, [1959].log_data[0].total := 300.0, [1959].log_data[0].time := 300.0,
        [1959].log_data[0].minminute := 35, [1959].log_data[0].maxminute := 35, [1959].log_data[0].valid := 1, [1959].log_data[1].valid := 1, [1959].log_data[2].valid := 1, [1959].log_data[3].valid := 1, [1959].log_data[4].valid := 1, [1959].log_data[5].valid := 1, [1959].log_data[6].valid := 1, [1959].log_data[7].valid := 1, [1959].log_data[8].valid := 1, [1959].log_data[9].valid := 1, [1959].log_data[10].valid := 1, [1959].log_data[11].valid := 1, [1959].log_data[12].valid := 1, [1959].log_data[13].valid := 1, [1959].log_data[14].valid := 1, [1959].log_data[15].valid := 1, [1959].log_data[16].valid := 1, [1959].log_data[17].valid := 1, [1959].log_data[18].valid := 1, [1959].log_data[19].valid := 1, [1959].time.Year := 2023, [1959].time.Month := 1, [1959].time.Day := 16, [1959].time.Hour := 11, [1959].time.Minute := 39, [1959].time.Second := 59, [1960].log_data[0].min := 1.0, [1960].log_data[0].max := 1.0, [1960].log_data[0].total := 300.0, [1960].log_data[0].time := 300.0, [1960].log_data[0].minminute := 40, [1960].log_data[0].maxminute := 40, [1960].log_data[0].valid := 1, [1960].log_data[1].valid := 1, [1960].log_data[2].valid := 1, [1960].log_data[3].valid := 1, [1960].log_data[4].valid := 1, [1960].log_data[5].valid := 1, [1960].log_data[6].valid := 1, [1960].log_data[7].valid := 1, [1960].log_data[8].valid := 1, [1960].log_data[9].valid := 1, [1960].log_data[10].valid := 1, [1960].log_data[11].valid := 1, [1960].log_data[12].valid := 1, [1960].log_data[13].valid := 1, [1960].log_data[14].valid := 1, [1960].log_data[15].valid := 1, [1960].log_data[16].valid := 1, [1960].log_data[17].valid := 1, [1960].log_data[18].valid := 1, [1960].log_data[19].valid := 1, [1960].time.Year := 2023, [1960].time.Month := 1, [1960].time.Day := 16, [1960].time.Hour := 11, [1960].time.Minute := 44, [1960].time.Second := 59,
        [1961].log_data[0].min := 1.0, [1961].log_data[0].max := 1.0, [1961].log_data[0].total := 300.0, [1961].log_data[0].time := 300.0, [1961].log_data[0].minminute := 45, [1961].log_data[0].maxminute := 45, [1961].log_data[0].valid := 1, [1961].log_data[1].valid := 1, [1961].log_data[2].valid := 1, [1961].log_data[3].valid := 1, [1961].log_data[4].valid := 1, [1961].log_data[5].valid := 1, [1961].log_data[6].valid := 1, [1961].log_data[7].valid := 1, [1961].log_data[8].valid := 1, [1961].log_data[9].valid := 1, [1961].log_data[10].valid := 1, [1961].log_data[11].valid := 1, [1961].log_data[12].valid := 1, [1961].log_data[13].valid := 1, [1961].log_data[14].valid := 1, [1961].log_data[15].valid := 1, [1961].log_data[16].valid := 1, [1961].log_data[17].valid := 1, [1961].log_data[18].valid := 1, [1961].log_data[19].valid := 1, [1961].time.Year := 2023, [1961].time.Month := 1, [1961].time.Day := 16, [1961].time.Hour := 11, [1961].time.Minute := 49, [1961].time.Second := 59, [1962].log_data[0].min := 1.0, [1962].log_data[0].max := 1.0, [1962].log_data[0].total := 300.0, [1962].log_data[0].time := 300.0, [1962].log_data[0].minminute := 50, [1962].log_data[0].maxminute := 50, [1962].log_data[0].valid := 1, [1962].log_data[1].valid := 1, [1962].log_data[2].valid := 1, [1962].log_data[3].valid := 1, [1962].log_data[4].valid := 1, [1962].log_data[5].valid := 1, [1962].log_data[6].valid := 1, [1962].log_data[7].valid := 1, [1962].log_data[8].valid := 1, [1962].log_data[9].valid := 1, [1962].log_data[10].valid := 1, [1962].log_data[11].valid := 1, [1962].log_data[12].valid := 1, [1962].log_data[13].valid := 1, [1962].log_data[14].valid := 1, [1962].log_data[15].valid := 1, [1962].log_data[16].valid := 1, [1962].log_data[17].valid := 1, [1962].log_data[18].valid := 1, [1962].log_data[19].valid := 1, [1962].time.Year := 2023, [1962].time.Month := 1,
        [1962].time.Day := 16, [1962].time.Hour := 11, [1962].time.Minute := 54, [1962].time.Second := 59, [1963].log_data[0].min := 1.0, [1963].log_data[0].max := 1.0, [1963].log_data[0].total := 300.0, [1963].log_data[0].time := 300.0, [1963].log_data[0].minminute := 55, [1963].log_data[0].maxminute := 55, [1963].log_data[0].valid := 1, [1963].log_data[1].valid := 1, [1963].log_data[2].valid := 1, [1963].log_data[3].valid := 1, [1963].log_data[4].valid := 1, [1963].log_data[5].valid := 1, [1963].log_data[6].valid := 1, [1963].log_data[7].valid := 1, [1963].log_data[8].valid := 1, [1963].log_data[9].valid := 1, [1963].log_data[10].valid := 1, [1963].log_data[11].valid := 1, [1963].log_data[12].valid := 1, [1963].log_data[13].valid := 1, [1963].log_data[14].valid := 1, [1963].log_data[15].valid := 1, [1963].log_data[16].valid := 1, [1963].log_data[17].valid := 1, [1963].log_data[18].valid := 1, [1963].log_data[19].valid := 1, [1963].time.Year := 2023, [1963].time.Month := 1, [1963].time.Day := 16, [1963].time.Hour := 11, [1963].time.Minute := 59, [1963].time.Second := 59, [1964].log_data[0].min := 1.0, [1964].log_data[0].max := 1.0, [1964].log_data[0].total := 300.0, [1964].log_data[0].time := 300.0, [1964].log_data[0].valid := 1, [1964].log_data[1].valid := 1, [1964].log_data[2].valid := 1, [1964].log_data[3].valid := 1, [1964].log_data[4].valid := 1, [1964].log_data[5].valid := 1, [1964].log_data[6].valid := 1, [1964].log_data[7].valid := 1, [1964].log_data[8].valid := 1, [1964].log_data[9].valid := 1, [1964].log_data[10].valid := 1, [1964].log_data[11].valid := 1, [1964].log_data[12].valid := 1, [1964].log_data[13].valid := 1, [1964].log_data[14].valid := 1, [1964].log_data[15].valid := 1, [1964].log_data[16].valid := 1, [1964].log_data[17].valid := 1, [1964].log_data[18].valid := 1, [1964].log_data[19].valid := 1,
        [1964].time.Year := 2023, [1964].time.Month := 1, [1964].time.Day := 16, [1964].time.Hour := 12, [1964].time.Minute := 4, [1964].time.Second := 59, [1965].log_data[0].min := 1.0, [1965].log_data[0].max := 1.0, [1965].log_data[0].total := 300.0, [1965].log_data[0].time := 300.0, [1965].log_data[0].minminute := 5, [1965].log_data[0].maxminute := 5, [1965].log_data[0].valid := 1, [1965].log_data[1].valid := 1, [1965].log_data[2].valid := 1, [1965].log_data[3].valid := 1, [1965].log_data[4].valid := 1, [1965].log_data[5].valid := 1, [1965].log_data[6].valid := 1, [1965].log_data[7].valid := 1, [1965].log_data[8].valid := 1, [1965].log_data[9].valid := 1, [1965].log_data[10].valid := 1, [1965].log_data[11].valid := 1, [1965].log_data[12].valid := 1, [1965].log_data[13].valid := 1, [1965].log_data[14].valid := 1, [1965].log_data[15].valid := 1, [1965].log_data[16].valid := 1, [1965].log_data[17].valid := 1, [1965].log_data[18].valid := 1, [1965].log_data[19].valid := 1, [1965].time.Year := 2023, [1965].time.Month := 1, [1965].time.Day := 16, [1965].time.Hour := 12, [1965].time.Minute := 9, [1965].time.Second := 59, [1966].log_data[0].min := 1.0, [1966].log_data[0].max := 1.0, [1966].log_data[0].total := 300.0, [1966].log_data[0].time := 300.0, [1966].log_data[0].minminute := 10, [1966].log_data[0].maxminute := 10, [1966].log_data[0].valid := 1, [1966].log_data[1].valid := 1, [1966].log_data[2].valid := 1, [1966].log_data[3].valid := 1, [1966].log_data[4].valid := 1, [1966].log_data[5].valid := 1, [1966].log_data[6].valid := 1, [1966].log_data[7].valid := 1, [1966].log_data[8].valid := 1, [1966].log_data[9].valid := 1, [1966].log_data[10].valid := 1, [1966].log_data[11].valid := 1, [1966].log_data[12].valid := 1, [1966].log_data[13].valid := 1, [1966].log_data[14].valid := 1, [1966].log_data[15].valid := 1,
        [1966].log_data[16].valid := 1, [1966].log_data[17].valid := 1, [1966].log_data[18].valid := 1, [1966].log_data[19].valid := 1, [1966].time.Year := 2023, [1966].time.Month := 1, [1966].time.Day := 16, [1966].time.Hour := 12, [1966].time.Minute := 14, [1966].time.Second := 59, [1967].log_data[0].min := 1.0, [1967].log_data[0].max := 1.0, [1967].log_data[0].total := 300.0, [1967].log_data[0].time := 300.0, [1967].log_data[0].minminute := 15, [1967].log_data[0].maxminute := 15, [1967].log_data[0].valid := 1, [1967].log_data[1].valid := 1, [1967].log_data[2].valid := 1, [1967].log_data[3].valid := 1, [1967].log_data[4].valid := 1, [1967].log_data[5].valid := 1, [1967].log_data[6].valid := 1, [1967].log_data[7].valid := 1, [1967].log_data[8].valid := 1, [1967].log_data[9].valid := 1, [1967].log_data[10].valid := 1, [1967].log_data[11].valid := 1, [1967].log_data[12].valid := 1, [1967].log_data[13].valid := 1, [1967].log_data[14].valid := 1, [1967].log_data[15].valid := 1, [1967].log_data[16].valid := 1, [1967].log_data[17].valid := 1, [1967].log_data[18].valid := 1, [1967].log_data[19].valid := 1, [1967].time.Year := 2023, [1967].time.Month := 1, [1967].time.Day := 16, [1967].time.Hour := 12, [1967].time.Minute := 19, [1967].time.Second := 59, [1968].log_data[0].min := 1.0, [1968].log_data[0].max := 1.0, [1968].log_data[0].total := 300.0, [1968].log_data[0].time := 300.0, [1968].log_data[0].minminute := 20, [1968].log_data[0].maxminute := 20, [1968].log_data[0].valid := 1, [1968].log_data[1].valid := 1, [1968].log_data[2].valid := 1, [1968].log_data[3].valid := 1, [1968].log_data[4].valid := 1, [1968].log_data[5].valid := 1, [1968].log_data[6].valid := 1, [1968].log_data[7].valid := 1, [1968].log_data[8].valid := 1, [1968].log_data[9].valid := 1, [1968].log_data[10].valid := 1, [1968].log_data[11].valid := 1,
        [1968].log_data[12].valid := 1, [1968].log_data[13].valid := 1, [1968].log_data[14].valid := 1, [1968].log_data[15].valid := 1, [1968].log_data[16].valid := 1, [1968].log_data[17].valid := 1, [1968].log_data[18].valid := 1, [1968].log_data[19].valid := 1, [1968].time.Year := 2023, [1968].time.Month := 1, [1968].time.Day := 16, [1968].time.Hour := 12, [1968].time.Minute := 24, [1968].time.Second := 59, [1969].log_data[0].min := 1.0, [1969].log_data[0].max := 1.0, [1969].log_data[0].total := 300.0, [1969].log_data[0].time := 300.0, [1969].log_data[0].minminute := 25, [1969].log_data[0].maxminute := 25, [1969].log_data[0].valid := 1, [1969].log_data[1].valid := 1, [1969].log_data[2].valid := 1, [1969].log_data[3].valid := 1, [1969].log_data[4].valid := 1, [1969].log_data[5].valid := 1, [1969].log_data[6].valid := 1, [1969].log_data[7].valid := 1, [1969].log_data[8].valid := 1, [1969].log_data[9].valid := 1, [1969].log_data[10].valid := 1, [1969].log_data[11].valid := 1, [1969].log_data[12].valid := 1, [1969].log_data[13].valid := 1, [1969].log_data[14].valid := 1, [1969].log_data[15].valid := 1, [1969].log_data[16].valid := 1, [1969].log_data[17].valid := 1, [1969].log_data[18].valid := 1, [1969].log_data[19].valid := 1, [1969].time.Year := 2023, [1969].time.Month := 1, [1969].time.Day := 16, [1969].time.Hour := 12, [1969].time.Minute := 29, [1969].time.Second := 59, [1970].log_data[0].min := 1.0, [1970].log_data[0].max := 1.0, [1970].log_data[0].total := 300.0, [1970].log_data[0].time := 300.0, [1970].log_data[0].minminute := 30, [1970].log_data[0].maxminute := 30, [1970].log_data[0].valid := 1, [1970].log_data[1].valid := 1, [1970].log_data[2].valid := 1, [1970].log_data[3].valid := 1, [1970].log_data[4].valid := 1, [1970].log_data[5].valid := 1, [1970].log_data[6].valid := 1, [1970].log_data[7].valid := 1,
        [1970].log_data[8].valid := 1, [1970].log_data[9].valid := 1, [1970].log_data[10].valid := 1, [1970].log_data[11].valid := 1, [1970].log_data[12].valid := 1, [1970].log_data[13].valid := 1, [1970].log_data[14].valid := 1, [1970].log_data[15].valid := 1, [1970].log_data[16].valid := 1, [1970].log_data[17].valid := 1, [1970].log_data[18].valid := 1, [1970].log_data[19].valid := 1, [1970].time.Year := 2023, [1970].time.Month := 1, [1970].time.Day := 16, [1970].time.Hour := 12, [1970].time.Minute := 34, [1970].time.Second := 59, [1971].log_data[0].min := 1.0, [1971].log_data[0].max := 1.0, [1971].log_data[0].total := 300.0, [1971].log_data[0].time := 300.0, [1971].log_data[0].minminute := 35, [1971].log_data[0].maxminute := 35, [1971].log_data[0].valid := 1, [1971].log_data[1].valid := 1, [1971].log_data[2].valid := 1, [1971].log_data[3].valid := 1, [1971].log_data[4].valid := 1, [1971].log_data[5].valid := 1, [1971].log_data[6].valid := 1, [1971].log_data[7].valid := 1, [1971].log_data[8].valid := 1, [1971].log_data[9].valid := 1, [1971].log_data[10].valid := 1, [1971].log_data[11].valid := 1, [1971].log_data[12].valid := 1, [1971].log_data[13].valid := 1, [1971].log_data[14].valid := 1, [1971].log_data[15].valid := 1, [1971].log_data[16].valid := 1, [1971].log_data[17].valid := 1, [1971].log_data[18].valid := 1, [1971].log_data[19].valid := 1, [1971].time.Year := 2023, [1971].time.Month := 1, [1971].time.Day := 16, [1971].time.Hour := 12, [1971].time.Minute := 39, [1971].time.Second := 59, [1972].log_data[0].min := 1.0, [1972].log_data[0].max := 1.0, [1972].log_data[0].total := 300.0, [1972].log_data[0].time := 300.0, [1972].log_data[0].minminute := 40, [1972].log_data[0].maxminute := 40, [1972].log_data[0].valid := 1, [1972].log_data[1].valid := 1, [1972].log_data[2].valid := 1, [1972].log_data[3].valid := 1,
        [1972].log_data[4].valid := 1, [1972].log_data[5].valid := 1, [1972].log_data[6].valid := 1, [1972].log_data[7].valid := 1, [1972].log_data[8].valid := 1, [1972].log_data[9].valid := 1, [1972].log_data[10].valid := 1, [1972].log_data[11].valid := 1, [1972].log_data[12].valid := 1, [1972].log_data[13].valid := 1, [1972].log_data[14].valid := 1, [1972].log_data[15].valid := 1, [1972].log_data[16].valid := 1, [1972].log_data[17].valid := 1, [1972].log_data[18].valid := 1, [1972].log_data[19].valid := 1, [1972].time.Year := 2023, [1972].time.Month := 1, [1972].time.Day := 16, [1972].time.Hour := 12, [1972].time.Minute := 44, [1972].time.Second := 59, [1973].log_data[0].min := 1.0, [1973].log_data[0].max := 1.0, [1973].log_data[0].total := 300.0, [1973].log_data[0].time := 300.0, [1973].log_data[0].minminute := 45, [1973].log_data[0].maxminute := 45, [1973].log_data[0].valid := 1, [1973].log_data[1].valid := 1, [1973].log_data[2].valid := 1, [1973].log_data[3].valid := 1, [1973].log_data[4].valid := 1, [1973].log_data[5].valid := 1, [1973].log_data[6].valid := 1, [1973].log_data[7].valid := 1, [1973].log_data[8].valid := 1, [1973].log_data[9].valid := 1, [1973].log_data[10].valid := 1, [1973].log_data[11].valid := 1, [1973].log_data[12].valid := 1, [1973].log_data[13].valid := 1, [1973].log_data[14].valid := 1, [1973].log_data[15].valid := 1, [1973].log_data[16].valid := 1, [1973].log_data[17].valid := 1, [1973].log_data[18].valid := 1, [1973].log_data[19].valid := 1, [1973].time.Year := 2023, [1973].time.Month := 1, [1973].time.Day := 16, [1973].time.Hour := 12, [1973].time.Minute := 49, [1973].time.Second := 59, [1974].log_data[0].min := 1.0, [1974].log_data[0].max := 1.0, [1974].log_data[0].total := 300.0, [1974].log_data[0].time := 300.0, [1974].log_data[0].minminute := 50, [1974].log_data[0].maxminute := 50,
        [1974].log_data[0].valid := 1, [1974].log_data[1].valid := 1, [1974].log_data[2].valid := 1, [1974].log_data[3].valid := 1, [1974].log_data[4].valid := 1, [1974].log_data[5].valid := 1, [1974].log_data[6].valid := 1, [1974].log_data[7].valid := 1, [1974].log_data[8].valid := 1, [1974].log_data[9].valid := 1, [1974].log_data[10].valid := 1, [1974].log_data[11].valid := 1, [1974].log_data[12].valid := 1, [1974].log_data[13].valid := 1, [1974].log_data[14].valid := 1, [1974].log_data[15].valid := 1, [1974].log_data[16].valid := 1, [1974].log_data[17].valid := 1, [1974].log_data[18].valid := 1, [1974].log_data[19].valid := 1, [1974].time.Year := 2023, [1974].time.Month := 1, [1974].time.Day := 16, [1974].time.Hour := 12, [1974].time.Minute := 54, [1974].time.Second := 59, [1975].log_data[0].min := 1.0, [1975].log_data[0].max := 1.0, [1975].log_data[0].total := 300.0, [1975].log_data[0].time := 300.0, [1975].log_data[0].minminute := 55, [1975].log_data[0].maxminute := 55, [1975].log_data[0].valid := 1, [1975].log_data[1].valid := 1, [1975].log_data[2].valid := 1, [1975].log_data[3].valid := 1, [1975].log_data[4].valid := 1, [1975].log_data[5].valid := 1, [1975].log_data[6].valid := 1, [1975].log_data[7].valid := 1, [1975].log_data[8].valid := 1, [1975].log_data[9].valid := 1, [1975].log_data[10].valid := 1, [1975].log_data[11].valid := 1, [1975].log_data[12].valid := 1, [1975].log_data[13].valid := 1, [1975].log_data[14].valid := 1, [1975].log_data[15].valid := 1, [1975].log_data[16].valid := 1, [1975].log_data[17].valid := 1, [1975].log_data[18].valid := 1, [1975].log_data[19].valid := 1, [1975].time.Year := 2023, [1975].time.Month := 1, [1975].time.Day := 16, [1975].time.Hour := 12, [1975].time.Minute := 59, [1975].time.Second := 59, [1976].log_data[0].min := 1.0, [1976].log_data[0].max := 1.0,
        [1976].log_data[0].total := 300.0, [1976].log_data[0].time := 300.0, [1976].log_data[0].valid := 1, [1976].log_data[1].valid := 1, [1976].log_data[2].valid := 1, [1976].log_data[3].valid := 1, [1976].log_data[4].valid := 1, [1976].log_data[5].valid := 1, [1976].log_data[6].valid := 1, [1976].log_data[7].valid := 1, [1976].log_data[8].valid := 1, [1976].log_data[9].valid := 1, [1976].log_data[10].valid := 1, [1976].log_data[11].valid := 1, [1976].log_data[12].valid := 1, [1976].log_data[13].valid := 1, [1976].log_data[14].valid := 1, [1976].log_data[15].valid := 1, [1976].log_data[16].valid := 1, [1976].log_data[17].valid := 1, [1976].log_data[18].valid := 1, [1976].log_data[19].valid := 1, [1976].time.Year := 2023, [1976].time.Month := 1, [1976].time.Day := 16, [1976].time.Hour := 13, [1976].time.Minute := 4, [1976].time.Second := 59, [1977].log_data[0].min := 1.0, [1977].log_data[0].max := 1.0, [1977].log_data[0].total := 300.0, [1977].log_data[0].time := 300.0, [1977].log_data[0].minminute := 5, [1977].log_data[0].maxminute := 5, [1977].log_data[0].valid := 1, [1977].log_data[1].valid := 1, [1977].log_data[2].valid := 1, [1977].log_data[3].valid := 1, [1977].log_data[4].valid := 1, [1977].log_data[5].valid := 1, [1977].log_data[6].valid := 1, [1977].log_data[7].valid := 1, [1977].log_data[8].valid := 1, [1977].log_data[9].valid := 1, [1977].log_data[10].valid := 1, [1977].log_data[11].valid := 1, [1977].log_data[12].valid := 1, [1977].log_data[13].valid := 1, [1977].log_data[14].valid := 1, [1977].log_data[15].valid := 1, [1977].log_data[16].valid := 1, [1977].log_data[17].valid := 1, [1977].log_data[18].valid := 1, [1977].log_data[19].valid := 1, [1977].time.Year := 2023, [1977].time.Month := 1, [1977].time.Day := 16, [1977].time.Hour := 13, [1977].time.Minute := 9, [1977].time.Second := 59,
        [1978].log_data[0].min := 1.0, [1978].log_data[0].max := 1.0, [1978].log_data[0].total := 300.0, [1978].log_data[0].time := 300.0, [1978].log_data[0].minminute := 10, [1978].log_data[0].maxminute := 10, [1978].log_data[0].valid := 1, [1978].log_data[1].valid := 1, [1978].log_data[2].valid := 1, [1978].log_data[3].valid := 1, [1978].log_data[4].valid := 1, [1978].log_data[5].valid := 1, [1978].log_data[6].valid := 1, [1978].log_data[7].valid := 1, [1978].log_data[8].valid := 1, [1978].log_data[9].valid := 1, [1978].log_data[10].valid := 1, [1978].log_data[11].valid := 1, [1978].log_data[12].valid := 1, [1978].log_data[13].valid := 1, [1978].log_data[14].valid := 1, [1978].log_data[15].valid := 1, [1978].log_data[16].valid := 1, [1978].log_data[17].valid := 1, [1978].log_data[18].valid := 1, [1978].log_data[19].valid := 1, [1978].time.Year := 2023, [1978].time.Month := 1, [1978].time.Day := 16, [1978].time.Hour := 13, [1978].time.Minute := 14, [1978].time.Second := 59, [1979].log_data[0].min := 1.0, [1979].log_data[0].max := 1.0, [1979].log_data[0].total := 300.0, [1979].log_data[0].time := 300.0, [1979].log_data[0].minminute := 15, [1979].log_data[0].maxminute := 15, [1979].log_data[0].valid := 1, [1979].log_data[1].valid := 1, [1979].log_data[2].valid := 1, [1979].log_data[3].valid := 1, [1979].log_data[4].valid := 1, [1979].log_data[5].valid := 1, [1979].log_data[6].valid := 1, [1979].log_data[7].valid := 1, [1979].log_data[8].valid := 1, [1979].log_data[9].valid := 1, [1979].log_data[10].valid := 1, [1979].log_data[11].valid := 1, [1979].log_data[12].valid := 1, [1979].log_data[13].valid := 1, [1979].log_data[14].valid := 1, [1979].log_data[15].valid := 1, [1979].log_data[16].valid := 1, [1979].log_data[17].valid := 1, [1979].log_data[18].valid := 1, [1979].log_data[19].valid := 1, [1979].time.Year := 2023, [1979].time.Month := 1,
        [1979].time.Day := 16, [1979].time.Hour := 13, [1979].time.Minute := 19, [1979].time.Second := 59, [1980].log_data[0].min := 1.0, [1980].log_data[0].max := 1.0, [1980].log_data[0].total := 300.0, [1980].log_data[0].time := 300.0, [1980].log_data[0].minminute := 20, [1980].log_data[0].maxminute := 20, [1980].log_data[0].valid := 1, [1980].log_data[1].valid := 1, [1980].log_data[2].valid := 1, [1980].log_data[3].valid := 1, [1980].log_data[4].valid := 1, [1980].log_data[5].valid := 1, [1980].log_data[6].valid := 1, [1980].log_data[7].valid := 1, [1980].log_data[8].valid := 1, [1980].log_data[9].valid := 1, [1980].log_data[10].valid := 1, [1980].log_data[11].valid := 1, [1980].log_data[12].valid := 1, [1980].log_data[13].valid := 1, [1980].log_data[14].valid := 1, [1980].log_data[15].valid := 1, [1980].log_data[16].valid := 1, [1980].log_data[17].valid := 1, [1980].log_data[18].valid := 1, [1980].log_data[19].valid := 1, [1980].time.Year := 2023, [1980].time.Month := 1, [1980].time.Day := 16, [1980].time.Hour := 13, [1980].time.Minute := 24, [1980].time.Second := 59, [1981].log_data[0].min := 1.0, [1981].log_data[0].max := 1.0, [1981].log_data[0].total := 300.0, [1981].log_data[0].time := 300.0, [1981].log_data[0].minminute := 25, [1981].log_data[0].maxminute := 25, [1981].log_data[0].valid := 1, [1981].log_data[1].valid := 1, [1981].log_data[2].valid := 1, [1981].log_data[3].valid := 1, [1981].log_data[4].valid := 1, [1981].log_data[5].valid := 1, [1981].log_data[6].valid := 1, [1981].log_data[7].valid := 1, [1981].log_data[8].valid := 1, [1981].log_data[9].valid := 1, [1981].log_data[10].valid := 1, [1981].log_data[11].valid := 1, [1981].log_data[12].valid := 1, [1981].log_data[13].valid := 1, [1981].log_data[14].valid := 1, [1981].log_data[15].valid := 1, [1981].log_data[16].valid := 1, [1981].log_data[17].valid := 1,
        [1981].log_data[18].valid := 1, [1981].log_data[19].valid := 1, [1981].time.Year := 2023, [1981].time.Month := 1, [1981].time.Day := 16, [1981].time.Hour := 13, [1981].time.Minute := 29, [1981].time.Second := 59, [1982].log_data[0].min := 1.0, [1982].log_data[0].max := 1.0, [1982].log_data[0].total := 300.0, [1982].log_data[0].time := 300.0, [1982].log_data[0].minminute := 30, [1982].log_data[0].maxminute := 30, [1982].log_data[0].valid := 1, [1982].log_data[1].valid := 1, [1982].log_data[2].valid := 1, [1982].log_data[3].valid := 1, [1982].log_data[4].valid := 1, [1982].log_data[5].valid := 1, [1982].log_data[6].valid := 1, [1982].log_data[7].valid := 1, [1982].log_data[8].valid := 1, [1982].log_data[9].valid := 1, [1982].log_data[10].valid := 1, [1982].log_data[11].valid := 1, [1982].log_data[12].valid := 1, [1982].log_data[13].valid := 1, [1982].log_data[14].valid := 1, [1982].log_data[15].valid := 1, [1982].log_data[16].valid := 1, [1982].log_data[17].valid := 1, [1982].log_data[18].valid := 1, [1982].log_data[19].valid := 1, [1982].time.Year := 2023, [1982].time.Month := 1, [1982].time.Day := 16, [1982].time.Hour := 13, [1982].time.Minute := 34, [1982].time.Second := 59, [1983].log_data[0].min := 1.0, [1983].log_data[0].max := 1.0, [1983].log_data[0].total := 300.0, [1983].log_data[0].time := 300.0, [1983].log_data[0].minminute := 35, [1983].log_data[0].maxminute := 35, [1983].log_data[0].valid := 1, [1983].log_data[1].valid := 1, [1983].log_data[2].valid := 1, [1983].log_data[3].valid := 1, [1983].log_data[4].valid := 1, [1983].log_data[5].valid := 1, [1983].log_data[6].valid := 1, [1983].log_data[7].valid := 1, [1983].log_data[8].valid := 1, [1983].log_data[9].valid := 1, [1983].log_data[10].valid := 1, [1983].log_data[11].valid := 1, [1983].log_data[12].valid := 1, [1983].log_data[13].valid := 1,
        [1983].log_data[14].valid := 1, [1983].log_data[15].valid := 1, [1983].log_data[16].valid := 1, [1983].log_data[17].valid := 1, [1983].log_data[18].valid := 1, [1983].log_data[19].valid := 1, [1983].time.Year := 2023, [1983].time.Month := 1, [1983].time.Day := 16, [1983].time.Hour := 13, [1983].time.Minute := 39, [1983].time.Second := 59, [1984].log_data[0].min := 1.0, [1984].log_data[0].max := 1.0, [1984].log_data[0].total := 300.0, [1984].log_data[0].time := 300.0, [1984].log_data[0].minminute := 40, [1984].log_data[0].maxminute := 40, [1984].log_data[0].valid := 1, [1984].log_data[1].valid := 1, [1984].log_data[2].valid := 1, [1984].log_data[3].valid := 1, [1984].log_data[4].valid := 1, [1984].log_data[5].valid := 1, [1984].log_data[6].valid := 1, [1984].log_data[7].valid := 1, [1984].log_data[8].valid := 1, [1984].log_data[9].valid := 1, [1984].log_data[10].valid := 1, [1984].log_data[11].valid := 1, [1984].log_data[12].valid := 1, [1984].log_data[13].valid := 1, [1984].log_data[14].valid := 1, [1984].log_data[15].valid := 1, [1984].log_data[16].valid := 1, [1984].log_data[17].valid := 1, [1984].log_data[18].valid := 1, [1984].log_data[19].valid := 1, [1984].time.Year := 2023, [1984].time.Month := 1, [1984].time.Day := 16, [1984].time.Hour := 13, [1984].time.Minute := 44, [1984].time.Second := 59, [1985].log_data[0].min := 1.0, [1985].log_data[0].max := 1.0, [1985].log_data[0].total := 300.0, [1985].log_data[0].time := 300.0, [1985].log_data[0].minminute := 45, [1985].log_data[0].maxminute := 45, [1985].log_data[0].valid := 1, [1985].log_data[1].valid := 1, [1985].log_data[2].valid := 1, [1985].log_data[3].valid := 1, [1985].log_data[4].valid := 1, [1985].log_data[5].valid := 1, [1985].log_data[6].valid := 1, [1985].log_data[7].valid := 1, [1985].log_data[8].valid := 1, [1985].log_data[9].valid := 1,
        [1985].log_data[10].valid := 1, [1985].log_data[11].valid := 1, [1985].log_data[12].valid := 1, [1985].log_data[13].valid := 1, [1985].log_data[14].valid := 1, [1985].log_data[15].valid := 1, [1985].log_data[16].valid := 1, [1985].log_data[17].valid := 1, [1985].log_data[18].valid := 1, [1985].log_data[19].valid := 1, [1985].time.Year := 2023, [1985].time.Month := 1, [1985].time.Day := 16, [1985].time.Hour := 13, [1985].time.Minute := 49, [1985].time.Second := 59, [1986].log_data[0].min := 1.0, [1986].log_data[0].max := 1.0, [1986].log_data[0].total := 300.0, [1986].log_data[0].time := 300.0, [1986].log_data[0].minminute := 50, [1986].log_data[0].maxminute := 50, [1986].log_data[0].valid := 1, [1986].log_data[1].valid := 1, [1986].log_data[2].valid := 1, [1986].log_data[3].valid := 1, [1986].log_data[4].valid := 1, [1986].log_data[5].valid := 1, [1986].log_data[6].valid := 1, [1986].log_data[7].valid := 1, [1986].log_data[8].valid := 1, [1986].log_data[9].valid := 1, [1986].log_data[10].valid := 1, [1986].log_data[11].valid := 1, [1986].log_data[12].valid := 1, [1986].log_data[13].valid := 1, [1986].log_data[14].valid := 1, [1986].log_data[15].valid := 1, [1986].log_data[16].valid := 1, [1986].log_data[17].valid := 1, [1986].log_data[18].valid := 1, [1986].log_data[19].valid := 1, [1986].time.Year := 2023, [1986].time.Month := 1, [1986].time.Day := 16, [1986].time.Hour := 13, [1986].time.Minute := 54, [1986].time.Second := 59, [1987].log_data[0].min := 1.0, [1987].log_data[0].max := 1.0, [1987].log_data[0].total := 300.0, [1987].log_data[0].time := 300.0, [1987].log_data[0].minminute := 55, [1987].log_data[0].maxminute := 55, [1987].log_data[0].valid := 1, [1987].log_data[1].valid := 1, [1987].log_data[2].valid := 1, [1987].log_data[3].valid := 1, [1987].log_data[4].valid := 1, [1987].log_data[5].valid := 1,
        [1987].log_data[6].valid := 1, [1987].log_data[7].valid := 1, [1987].log_data[8].valid := 1, [1987].log_data[9].valid := 1, [1987].log_data[10].valid := 1, [1987].log_data[11].valid := 1, [1987].log_data[12].valid := 1, [1987].log_data[13].valid := 1, [1987].log_data[14].valid := 1, [1987].log_data[15].valid := 1, [1987].log_data[16].valid := 1, [1987].log_data[17].valid := 1, [1987].log_data[18].valid := 1, [1987].log_data[19].valid := 1, [1987].time.Year := 2023, [1987].time.Month := 1, [1987].time.Day := 16, [1987].time.Hour := 13, [1987].time.Minute := 59, [1987].time.Second := 59, [1988].log_data[0].min := 1.0, [1988].log_data[0].max := 1.0, [1988].log_data[0].total := 300.0, [1988].log_data[0].time := 300.0, [1988].log_data[0].valid := 1, [1988].log_data[1].valid := 1, [1988].log_data[2].valid := 1, [1988].log_data[3].valid := 1, [1988].log_data[4].valid := 1, [1988].log_data[5].valid := 1, [1988].log_data[6].valid := 1, [1988].log_data[7].valid := 1, [1988].log_data[8].valid := 1, [1988].log_data[9].valid := 1, [1988].log_data[10].valid := 1, [1988].log_data[11].valid := 1, [1988].log_data[12].valid := 1, [1988].log_data[13].valid := 1, [1988].log_data[14].valid := 1, [1988].log_data[15].valid := 1, [1988].log_data[16].valid := 1, [1988].log_data[17].valid := 1, [1988].log_data[18].valid := 1, [1988].log_data[19].valid := 1, [1988].time.Year := 2023, [1988].time.Month := 1, [1988].time.Day := 16, [1988].time.Hour := 14, [1988].time.Minute := 4, [1988].time.Second := 59, [1989].log_data[0].min := 1.0, [1989].log_data[0].max := 1.0, [1989].log_data[0].total := 300.0, [1989].log_data[0].time := 300.0, [1989].log_data[0].minminute := 5, [1989].log_data[0].maxminute := 5, [1989].log_data[0].valid := 1, [1989].log_data[1].valid := 1, [1989].log_data[2].valid := 1, [1989].log_data[3].valid := 1,
        [1989].log_data[4].valid := 1, [1989].log_data[5].valid := 1, [1989].log_data[6].valid := 1, [1989].log_data[7].valid := 1, [1989].log_data[8].valid := 1, [1989].log_data[9].valid := 1, [1989].log_data[10].valid := 1, [1989].log_data[11].valid := 1, [1989].log_data[12].valid := 1, [1989].log_data[13].valid := 1, [1989].log_data[14].valid := 1, [1989].log_data[15].valid := 1, [1989].log_data[16].valid := 1, [1989].log_data[17].valid := 1, [1989].log_data[18].valid := 1, [1989].log_data[19].valid := 1, [1989].time.Year := 2023, [1989].time.Month := 1, [1989].time.Day := 16, [1989].time.Hour := 14, [1989].time.Minute := 9, [1989].time.Second := 59, [1990].log_data[0].min := 1.0, [1990].log_data[0].max := 1.0, [1990].log_data[0].total := 300.0, [1990].log_data[0].time := 300.0, [1990].log_data[0].minminute := 10, [1990].log_data[0].maxminute := 10, [1990].log_data[0].valid := 1, [1990].log_data[1].valid := 1, [1990].log_data[2].valid := 1, [1990].log_data[3].valid := 1, [1990].log_data[4].valid := 1, [1990].log_data[5].valid := 1, [1990].log_data[6].valid := 1, [1990].log_data[7].valid := 1, [1990].log_data[8].valid := 1, [1990].log_data[9].valid := 1, [1990].log_data[10].valid := 1, [1990].log_data[11].valid := 1, [1990].log_data[12].valid := 1, [1990].log_data[13].valid := 1, [1990].log_data[14].valid := 1, [1990].log_data[15].valid := 1, [1990].log_data[16].valid := 1, [1990].log_data[17].valid := 1, [1990].log_data[18].valid := 1, [1990].log_data[19].valid := 1, [1990].time.Year := 2023, [1990].time.Month := 1, [1990].time.Day := 16, [1990].time.Hour := 14, [1990].time.Minute := 14, [1990].time.Second := 59, [1991].log_data[0].min := 1.0, [1991].log_data[0].max := 1.0, [1991].log_data[0].total := 300.0, [1991].log_data[0].time := 300.0, [1991].log_data[0].minminute := 15, [1991].log_data[0].maxminute := 15,
        [1991].log_data[0].valid := 1, [1991].log_data[1].valid := 1, [1991].log_data[2].valid := 1, [1991].log_data[3].valid := 1, [1991].log_data[4].valid := 1, [1991].log_data[5].valid := 1, [1991].log_data[6].valid := 1, [1991].log_data[7].valid := 1, [1991].log_data[8].valid := 1, [1991].log_data[9].valid := 1, [1991].log_data[10].valid := 1, [1991].log_data[11].valid := 1, [1991].log_data[12].valid := 1, [1991].log_data[13].valid := 1, [1991].log_data[14].valid := 1, [1991].log_data[15].valid := 1, [1991].log_data[16].valid := 1, [1991].log_data[17].valid := 1, [1991].log_data[18].valid := 1, [1991].log_data[19].valid := 1, [1991].time.Year := 2023, [1991].time.Month := 1, [1991].time.Day := 16, [1991].time.Hour := 14, [1991].time.Minute := 19, [1991].time.Second := 59, [1992].log_data[0].min := 1.0, [1992].log_data[0].max := 1.0, [1992].log_data[0].total := 300.0, [1992].log_data[0].time := 300.0, [1992].log_data[0].minminute := 20, [1992].log_data[0].maxminute := 20, [1992].log_data[0].valid := 1, [1992].log_data[1].valid := 1, [1992].log_data[2].valid := 1, [1992].log_data[3].valid := 1, [1992].log_data[4].valid := 1, [1992].log_data[5].valid := 1, [1992].log_data[6].valid := 1, [1992].log_data[7].valid := 1, [1992].log_data[8].valid := 1, [1992].log_data[9].valid := 1, [1992].log_data[10].valid := 1, [1992].log_data[11].valid := 1, [1992].log_data[12].valid := 1, [1992].log_data[13].valid := 1, [1992].log_data[14].valid := 1, [1992].log_data[15].valid := 1, [1992].log_data[16].valid := 1, [1992].log_data[17].valid := 1, [1992].log_data[18].valid := 1, [1992].log_data[19].valid := 1, [1992].time.Year := 2023, [1992].time.Month := 1, [1992].time.Day := 16, [1992].time.Hour := 14, [1992].time.Minute := 24, [1992].time.Second := 59, [1993].log_data[0].min := 1.0, [1993].log_data[0].max := 1.0,
        [1993].log_data[0].total := 300.0, [1993].log_data[0].time := 300.0, [1993].log_data[0].minminute := 25, [1993].log_data[0].maxminute := 25, [1993].log_data[0].valid := 1, [1993].log_data[1].valid := 1, [1993].log_data[2].valid := 1, [1993].log_data[3].valid := 1, [1993].log_data[4].valid := 1, [1993].log_data[5].valid := 1, [1993].log_data[6].valid := 1, [1993].log_data[7].valid := 1, [1993].log_data[8].valid := 1, [1993].log_data[9].valid := 1, [1993].log_data[10].valid := 1, [1993].log_data[11].valid := 1, [1993].log_data[12].valid := 1, [1993].log_data[13].valid := 1, [1993].log_data[14].valid := 1, [1993].log_data[15].valid := 1, [1993].log_data[16].valid := 1, [1993].log_data[17].valid := 1, [1993].log_data[18].valid := 1, [1993].log_data[19].valid := 1, [1993].time.Year := 2023, [1993].time.Month := 1, [1993].time.Day := 16, [1993].time.Hour := 14, [1993].time.Minute := 29, [1993].time.Second := 59, [1994].log_data[0].min := 1.0, [1994].log_data[0].max := 1.0, [1994].log_data[0].total := 300.0, [1994].log_data[0].time := 300.0, [1994].log_data[0].minminute := 30, [1994].log_data[0].maxminute := 30, [1994].log_data[0].valid := 1, [1994].log_data[1].valid := 1, [1994].log_data[2].valid := 1, [1994].log_data[3].valid := 1, [1994].log_data[4].valid := 1, [1994].log_data[5].valid := 1, [1994].log_data[6].valid := 1, [1994].log_data[7].valid := 1, [1994].log_data[8].valid := 1, [1994].log_data[9].valid := 1, [1994].log_data[10].valid := 1, [1994].log_data[11].valid := 1, [1994].log_data[12].valid := 1, [1994].log_data[13].valid := 1, [1994].log_data[14].valid := 1, [1994].log_data[15].valid := 1, [1994].log_data[16].valid := 1, [1994].log_data[17].valid := 1, [1994].log_data[18].valid := 1, [1994].log_data[19].valid := 1, [1994].time.Year := 2023, [1994].time.Month := 1, [1994].time.Day := 16, [1994].time.Hour := 14,
        [1994].time.Minute := 34, [1994].time.Second := 59, [1995].log_data[0].min := 1.0, [1995].log_data[0].max := 1.0, [1995].log_data[0].total := 300.0, [1995].log_data[0].time := 300.0, [1995].log_data[0].minminute := 35, [1995].log_data[0].maxminute := 35, [1995].log_data[0].valid := 1, [1995].log_data[1].valid := 1, [1995].log_data[2].valid := 1, [1995].log_data[3].valid := 1, [1995].log_data[4].valid := 1, [1995].log_data[5].valid := 1, [1995].log_data[6].valid := 1, [1995].log_data[7].valid := 1, [1995].log_data[8].valid := 1, [1995].log_data[9].valid := 1, [1995].log_data[10].valid := 1, [1995].log_data[11].valid := 1, [1995].log_data[12].valid := 1, [1995].log_data[13].valid := 1, [1995].log_data[14].valid := 1, [1995].log_data[15].valid := 1, [1995].log_data[16].valid := 1, [1995].log_data[17].valid := 1, [1995].log_data[18].valid := 1, [1995].log_data[19].valid := 1, [1995].time.Year := 2023, [1995].time.Month := 1, [1995].time.Day := 16, [1995].time.Hour := 14, [1995].time.Minute := 39, [1995].time.Second := 59, [1996].log_data[0].min := 1.0, [1996].log_data[0].max := 1.0, [1996].log_data[0].total := 300.0, [1996].log_data[0].time := 300.0, [1996].log_data[0].minminute := 40, [1996].log_data[0].maxminute := 40, [1996].log_data[0].valid := 1, [1996].log_data[1].valid := 1, [1996].log_data[2].valid := 1, [1996].log_data[3].valid := 1, [1996].log_data[4].valid := 1, [1996].log_data[5].valid := 1, [1996].log_data[6].valid := 1, [1996].log_data[7].valid := 1, [1996].log_data[8].valid := 1, [1996].log_data[9].valid := 1, [1996].log_data[10].valid := 1, [1996].log_data[11].valid := 1, [1996].log_data[12].valid := 1, [1996].log_data[13].valid := 1, [1996].log_data[14].valid := 1, [1996].log_data[15].valid := 1, [1996].log_data[16].valid := 1, [1996].log_data[17].valid := 1, [1996].log_data[18].valid := 1, [1996].log_data[19].valid := 1,
        [1996].time.Year := 2023, [1996].time.Month := 1, [1996].time.Day := 16, [1996].time.Hour := 14, [1996].time.Minute := 44, [1996].time.Second := 59, [1997].log_data[0].min := 1.0, [1997].log_data[0].max := 1.0, [1997].log_data[0].total := 300.0, [1997].log_data[0].time := 300.0, [1997].log_data[0].minminute := 45, [1997].log_data[0].maxminute := 45, [1997].log_data[0].valid := 1, [1997].log_data[1].valid := 1, [1997].log_data[2].valid := 1, [1997].log_data[3].valid := 1, [1997].log_data[4].valid := 1, [1997].log_data[5].valid := 1, [1997].log_data[6].valid := 1, [1997].log_data[7].valid := 1, [1997].log_data[8].valid := 1, [1997].log_data[9].valid := 1, [1997].log_data[10].valid := 1, [1997].log_data[11].valid := 1, [1997].log_data[12].valid := 1, [1997].log_data[13].valid := 1, [1997].log_data[14].valid := 1, [1997].log_data[15].valid := 1, [1997].log_data[16].valid := 1, [1997].log_data[17].valid := 1, [1997].log_data[18].valid := 1, [1997].log_data[19].valid := 1, [1997].time.Year := 2023, [1997].time.Month := 1, [1997].time.Day := 16, [1997].time.Hour := 14, [1997].time.Minute := 49, [1997].time.Second := 59, [1998].log_data[0].min := 1.0, [1998].log_data[0].max := 1.0, [1998].log_data[0].total := 300.0, [1998].log_data[0].time := 300.0, [1998].log_data[0].minminute := 50, [1998].log_data[0].maxminute := 50, [1998].log_data[0].valid := 1, [1998].log_data[1].valid := 1, [1998].log_data[2].valid := 1, [1998].log_data[3].valid := 1, [1998].log_data[4].valid := 1, [1998].log_data[5].valid := 1, [1998].log_data[6].valid := 1, [1998].log_data[7].valid := 1, [1998].log_data[8].valid := 1, [1998].log_data[9].valid := 1, [1998].log_data[10].valid := 1, [1998].log_data[11].valid := 1, [1998].log_data[12].valid := 1, [1998].log_data[13].valid := 1, [1998].log_data[14].valid := 1, [1998].log_data[15].valid := 1,
        [1998].log_data[16].valid := 1, [1998].log_data[17].valid := 1, [1998].log_data[18].valid := 1, [1998].log_data[19].valid := 1, [1998].time.Year := 2023, [1998].time.Month := 1, [1998].time.Day := 16, [1998].time.Hour := 14, [1998].time.Minute := 54, [1998].time.Second := 59, [1999].log_data[0].min := 1.0, [1999].log_data[0].max := 1.0, [1999].log_data[0].total := 300.0, [1999].log_data[0].time := 300.0, [1999].log_data[0].minminute := 55, [1999].log_data[0].maxminute := 55, [1999].log_data[0].valid := 1, [1999].log_data[1].valid := 1, [1999].log_data[2].valid := 1, [1999].log_data[3].valid := 1, [1999].log_data[4].valid := 1, [1999].log_data[5].valid := 1, [1999].log_data[6].valid := 1, [1999].log_data[7].valid := 1, [1999].log_data[8].valid := 1, [1999].log_data[9].valid := 1, [1999].log_data[10].valid := 1, [1999].log_data[11].valid := 1, [1999].log_data[12].valid := 1, [1999].log_data[13].valid := 1, [1999].log_data[14].valid := 1, [1999].log_data[15].valid := 1, [1999].log_data[16].valid := 1, [1999].log_data[17].valid := 1, [1999].log_data[18].valid := 1, [1999].log_data[19].valid := 1, [1999].time.Year := 2023, [1999].time.Month := 1, [1999].time.Day := 16, [1999].time.Hour := 14, [1999].time.Minute := 59, [1999].time.Second := 59, [2000].log_data[0].min := 1.0, [2000].log_data[0].max := 1.0, [2000].log_data[0].total := 300.0, [2000].log_data[0].time := 300.0, [2000].log_data[0].valid := 1, [2000].log_data[1].valid := 1, [2000].log_data[2].valid := 1, [2000].log_data[3].valid := 1, [2000].log_data[4].valid := 1, [2000].log_data[5].valid := 1, [2000].log_data[6].valid := 1, [2000].log_data[7].valid := 1, [2000].log_data[8].valid := 1, [2000].log_data[9].valid := 1, [2000].log_data[10].valid := 1, [2000].log_data[11].valid := 1, [2000].log_data[12].valid := 1, [2000].log_data[13].valid := 1,
        [2000].log_data[14].valid := 1, [2000].log_data[15].valid := 1, [2000].log_data[16].valid := 1, [2000].log_data[17].valid := 1, [2000].log_data[18].valid := 1, [2000].log_data[19].valid := 1, [2000].time.Year := 2023, [2000].time.Month := 1, [2000].time.Day := 16, [2000].time.Hour := 15, [2000].time.Minute := 4, [2000].time.Second := 59, [2001].log_data[0].min := 1.0, [2001].log_data[0].max := 1.0, [2001].log_data[0].total := 300.0, [2001].log_data[0].time := 300.0, [2001].log_data[0].minminute := 5, [2001].log_data[0].maxminute := 5, [2001].log_data[0].valid := 1, [2001].log_data[1].valid := 1, [2001].log_data[2].valid := 1, [2001].log_data[3].valid := 1, [2001].log_data[4].valid := 1, [2001].log_data[5].valid := 1, [2001].log_data[6].valid := 1, [2001].log_data[7].valid := 1, [2001].log_data[8].valid := 1, [2001].log_data[9].valid := 1, [2001].log_data[10].valid := 1, [2001].log_data[11].valid := 1, [2001].log_data[12].valid := 1, [2001].log_data[13].valid := 1, [2001].log_data[14].valid := 1, [2001].log_data[15].valid := 1, [2001].log_data[16].valid := 1, [2001].log_data[17].valid := 1, [2001].log_data[18].valid := 1, [2001].log_data[19].valid := 1, [2001].time.Year := 2023, [2001].time.Month := 1, [2001].time.Day := 16, [2001].time.Hour := 15, [2001].time.Minute := 9, [2001].time.Second := 59, [2002].log_data[0].min := 1.0, [2002].log_data[0].max := 1.0, [2002].log_data[0].total := 300.0, [2002].log_data[0].time := 300.0, [2002].log_data[0].minminute := 10, [2002].log_data[0].maxminute := 10, [2002].log_data[0].valid := 1, [2002].log_data[1].valid := 1, [2002].log_data[2].valid := 1, [2002].log_data[3].valid := 1, [2002].log_data[4].valid := 1, [2002].log_data[5].valid := 1, [2002].log_data[6].valid := 1, [2002].log_data[7].valid := 1, [2002].log_data[8].valid := 1, [2002].log_data[9].valid := 1,
        [2002].log_data[10].valid := 1, [2002].log_data[11].valid := 1, [2002].log_data[12].valid := 1, [2002].log_data[13].valid := 1, [2002].log_data[14].valid := 1, [2002].log_data[15].valid := 1, [2002].log_data[16].valid := 1, [2002].log_data[17].valid := 1, [2002].log_data[18].valid := 1, [2002].log_data[19].valid := 1, [2002].time.Year := 2023, [2002].time.Month := 1, [2002].time.Day := 16, [2002].time.Hour := 15, [2002].time.Minute := 14, [2002].time.Second := 59, [2003].log_data[0].min := 1.0, [2003].log_data[0].max := 1.0, [2003].log_data[0].total := 300.0, [2003].log_data[0].time := 300.0, [2003].log_data[0].minminute := 15, [2003].log_data[0].maxminute := 15, [2003].log_data[0].valid := 1, [2003].log_data[1].valid := 1, [2003].log_data[2].valid := 1, [2003].log_data[3].valid := 1, [2003].log_data[4].valid := 1, [2003].log_data[5].valid := 1, [2003].log_data[6].valid := 1, [2003].log_data[7].valid := 1, [2003].log_data[8].valid := 1, [2003].log_data[9].valid := 1, [2003].log_data[10].valid := 1, [2003].log_data[11].valid := 1, [2003].log_data[12].valid := 1, [2003].log_data[13].valid := 1, [2003].log_data[14].valid := 1, [2003].log_data[15].valid := 1, [2003].log_data[16].valid := 1, [2003].log_data[17].valid := 1, [2003].log_data[18].valid := 1, [2003].log_data[19].valid := 1, [2003].time.Year := 2023, [2003].time.Month := 1, [2003].time.Day := 16, [2003].time.Hour := 15, [2003].time.Minute := 19, [2003].time.Second := 59, [2004].log_data[0].min := 1.0, [2004].log_data[0].max := 1.0, [2004].log_data[0].total := 300.0, [2004].log_data[0].time := 300.0, [2004].log_data[0].minminute := 20, [2004].log_data[0].maxminute := 20, [2004].log_data[0].valid := 1, [2004].log_data[1].valid := 1, [2004].log_data[2].valid := 1, [2004].log_data[3].valid := 1, [2004].log_data[4].valid := 1, [2004].log_data[5].valid := 1,
        [2004].log_data[6].valid := 1, [2004].log_data[7].valid := 1, [2004].log_data[8].valid := 1, [2004].log_data[9].valid := 1, [2004].log_data[10].valid := 1, [2004].log_data[11].valid := 1, [2004].log_data[12].valid := 1, [2004].log_data[13].valid := 1, [2004].log_data[14].valid := 1, [2004].log_data[15].valid := 1, [2004].log_data[16].valid := 1, [2004].log_data[17].valid := 1, [2004].log_data[18].valid := 1, [2004].log_data[19].valid := 1, [2004].time.Year := 2023, [2004].time.Month := 1, [2004].time.Day := 16, [2004].time.Hour := 15, [2004].time.Minute := 24, [2004].time.Second := 59, [2005].log_data[0].min := 1.0, [2005].log_data[0].max := 1.0, [2005].log_data[0].total := 300.0, [2005].log_data[0].time := 300.0, [2005].log_data[0].minminute := 25, [2005].log_data[0].maxminute := 25, [2005].log_data[0].valid := 1, [2005].log_data[1].valid := 1, [2005].log_data[2].valid := 1, [2005].log_data[3].valid := 1, [2005].log_data[4].valid := 1, [2005].log_data[5].valid := 1, [2005].log_data[6].valid := 1, [2005].log_data[7].valid := 1, [2005].log_data[8].valid := 1, [2005].log_data[9].valid := 1, [2005].log_data[10].valid := 1, [2005].log_data[11].valid := 1, [2005].log_data[12].valid := 1, [2005].log_data[13].valid := 1, [2005].log_data[14].valid := 1, [2005].log_data[15].valid := 1, [2005].log_data[16].valid := 1, [2005].log_data[17].valid := 1, [2005].log_data[18].valid := 1, [2005].log_data[19].valid := 1, [2005].time.Year := 2023, [2005].time.Month := 1, [2005].time.Day := 16, [2005].time.Hour := 15, [2005].time.Minute := 29, [2005].time.Second := 59, [2006].log_data[0].min := 1.0, [2006].log_data[0].max := 1.0, [2006].log_data[0].total := 300.0, [2006].log_data[0].time := 300.0, [2006].log_data[0].minminute := 30, [2006].log_data[0].maxminute := 30, [2006].log_data[0].valid := 1, [2006].log_data[1].valid := 1,
        [2006].log_data[2].valid := 1, [2006].log_data[3].valid := 1, [2006].log_data[4].valid := 1, [2006].log_data[5].valid := 1, [2006].log_data[6].valid := 1, [2006].log_data[7].valid := 1, [2006].log_data[8].valid := 1, [2006].log_data[9].valid := 1, [2006].log_data[10].valid := 1, [2006].log_data[11].valid := 1, [2006].log_data[12].valid := 1, [2006].log_data[13].valid := 1, [2006].log_data[14].valid := 1, [2006].log_data[15].valid := 1, [2006].log_data[16].valid := 1, [2006].log_data[17].valid := 1, [2006].log_data[18].valid := 1, [2006].log_data[19].valid := 1, [2006].time.Year := 2023, [2006].time.Month := 1, [2006].time.Day := 16, [2006].time.Hour := 15, [2006].time.Minute := 34, [2006].time.Second := 59, [2007].log_data[0].min := 1.0, [2007].log_data[0].max := 1.0, [2007].log_data[0].total := 300.0, [2007].log_data[0].time := 300.0, [2007].log_data[0].minminute := 35, [2007].log_data[0].maxminute := 35, [2007].log_data[0].valid := 1, [2007].log_data[1].valid := 1, [2007].log_data[2].valid := 1, [2007].log_data[3].valid := 1, [2007].log_data[4].valid := 1, [2007].log_data[5].valid := 1, [2007].log_data[6].valid := 1, [2007].log_data[7].valid := 1, [2007].log_data[8].valid := 1, [2007].log_data[9].valid := 1, [2007].log_data[10].valid := 1, [2007].log_data[11].valid := 1, [2007].log_data[12].valid := 1, [2007].log_data[13].valid := 1, [2007].log_data[14].valid := 1, [2007].log_data[15].valid := 1, [2007].log_data[16].valid := 1, [2007].log_data[17].valid := 1, [2007].log_data[18].valid := 1, [2007].log_data[19].valid := 1, [2007].time.Year := 2023, [2007].time.Month := 1, [2007].time.Day := 16, [2007].time.Hour := 15, [2007].time.Minute := 39, [2007].time.Second := 59, [2008].log_data[0].min := 1.0, [2008].log_data[0].max := 1.0, [2008].log_data[0].total := 300.0, [2008].log_data[0].time := 300.0,
        [2008].log_data[0].minminute := 40, [2008].log_data[0].maxminute := 40, [2008].log_data[0].valid := 1, [2008].log_data[1].valid := 1, [2008].log_data[2].valid := 1, [2008].log_data[3].valid := 1, [2008].log_data[4].valid := 1, [2008].log_data[5].valid := 1, [2008].log_data[6].valid := 1, [2008].log_data[7].valid := 1, [2008].log_data[8].valid := 1, [2008].log_data[9].valid := 1, [2008].log_data[10].valid := 1, [2008].log_data[11].valid := 1, [2008].log_data[12].valid := 1, [2008].log_data[13].valid := 1, [2008].log_data[14].valid := 1, [2008].log_data[15].valid := 1, [2008].log_data[16].valid := 1, [2008].log_data[17].valid := 1, [2008].log_data[18].valid := 1, [2008].log_data[19].valid := 1, [2008].time.Year := 2023, [2008].time.Month := 1, [2008].time.Day := 16, [2008].time.Hour := 15, [2008].time.Minute := 44, [2008].time.Second := 59, [2009].log_data[0].min := 1.0, [2009].log_data[0].max := 1.0, [2009].log_data[0].total := 300.0, [2009].log_data[0].time := 300.0, [2009].log_data[0].minminute := 45, [2009].log_data[0].maxminute := 45, [2009].log_data[0].valid := 1, [2009].log_data[1].valid := 1, [2009].log_data[2].valid := 1, [2009].log_data[3].valid := 1, [2009].log_data[4].valid := 1, [2009].log_data[5].valid := 1, [2009].log_data[6].valid := 1, [2009].log_data[7].valid := 1, [2009].log_data[8].valid := 1, [2009].log_data[9].valid := 1, [2009].log_data[10].valid := 1, [2009].log_data[11].valid := 1, [2009].log_data[12].valid := 1, [2009].log_data[13].valid := 1, [2009].log_data[14].valid := 1, [2009].log_data[15].valid := 1, [2009].log_data[16].valid := 1, [2009].log_data[17].valid := 1, [2009].log_data[18].valid := 1, [2009].log_data[19].valid := 1, [2009].time.Year := 2023, [2009].time.Month := 1, [2009].time.Day := 16, [2009].time.Hour := 15, [2009].time.Minute := 49, [2009].time.Second := 59,
        [2010].log_data[0].min := 1.0, [2010].log_data[0].max := 1.0, [2010].log_data[0].total := 300.0, [2010].log_data[0].time := 300.0, [2010].log_data[0].minminute := 50, [2010].log_data[0].maxminute := 50, [2010].log_data[0].valid := 1, [2010].log_data[1].valid := 1, [2010].log_data[2].valid := 1, [2010].log_data[3].valid := 1, [2010].log_data[4].valid := 1, [2010].log_data[5].valid := 1, [2010].log_data[6].valid := 1, [2010].log_data[7].valid := 1, [2010].log_data[8].valid := 1, [2010].log_data[9].valid := 1, [2010].log_data[10].valid := 1, [2010].log_data[11].valid := 1, [2010].log_data[12].valid := 1, [2010].log_data[13].valid := 1, [2010].log_data[14].valid := 1, [2010].log_data[15].valid := 1, [2010].log_data[16].valid := 1, [2010].log_data[17].valid := 1, [2010].log_data[18].valid := 1, [2010].log_data[19].valid := 1, [2010].time.Year := 2023, [2010].time.Month := 1, [2010].time.Day := 16, [2010].time.Hour := 15, [2010].time.Minute := 54, [2010].time.Second := 59, [2011].log_data[0].min := 1.0, [2011].log_data[0].max := 1.0, [2011].log_data[0].total := 300.0, [2011].log_data[0].time := 300.0, [2011].log_data[0].minminute := 55, [2011].log_data[0].maxminute := 55, [2011].log_data[0].valid := 1, [2011].log_data[1].valid := 1, [2011].log_data[2].valid := 1, [2011].log_data[3].valid := 1, [2011].log_data[4].valid := 1, [2011].log_data[5].valid := 1, [2011].log_data[6].valid := 1, [2011].log_data[7].valid := 1, [2011].log_data[8].valid := 1, [2011].log_data[9].valid := 1, [2011].log_data[10].valid := 1, [2011].log_data[11].valid := 1, [2011].log_data[12].valid := 1, [2011].log_data[13].valid := 1, [2011].log_data[14].valid := 1, [2011].log_data[15].valid := 1, [2011].log_data[16].valid := 1, [2011].log_data[17].valid := 1, [2011].log_data[18].valid := 1, [2011].log_data[19].valid := 1, [2011].time.Year := 2023, [2011].time.Month := 1,
        [2011].time.Day := 16, [2011].time.Hour := 15, [2011].time.Minute := 59, [2011].time.Second := 59, [2012].log_data[0].min := 1.0, [2012].log_data[0].max := 1.0, [2012].log_data[0].total := 300.0, [2012].log_data[0].time := 300.0, [2012].log_data[0].valid := 1, [2012].log_data[1].valid := 1, [2012].log_data[2].valid := 1, [2012].log_data[3].valid := 1, [2012].log_data[4].valid := 1, [2012].log_data[5].valid := 1, [2012].log_data[6].valid := 1, [2012].log_data[7].valid := 1, [2012].log_data[8].valid := 1, [2012].log_data[9].valid := 1, [2012].log_data[10].valid := 1, [2012].log_data[11].valid := 1, [2012].log_data[12].valid := 1, [2012].log_data[13].valid := 1, [2012].log_data[14].valid := 1, [2012].log_data[15].valid := 1, [2012].log_data[16].valid := 1, [2012].log_data[17].valid := 1, [2012].log_data[18].valid := 1, [2012].log_data[19].valid := 1, [2012].time.Year := 2023, [2012].time.Month := 1, [2012].time.Day := 16, [2012].time.Hour := 16, [2012].time.Minute := 4, [2012].time.Second := 59, [2013].log_data[0].min := 1.0, [2013].log_data[0].max := 1.0, [2013].log_data[0].total := 300.0, [2013].log_data[0].time := 300.0, [2013].log_data[0].minminute := 5, [2013].log_data[0].maxminute := 5, [2013].log_data[0].valid := 1, [2013].log_data[1].valid := 1, [2013].log_data[2].valid := 1, [2013].log_data[3].valid := 1, [2013].log_data[4].valid := 1, [2013].log_data[5].valid := 1, [2013].log_data[6].valid := 1, [2013].log_data[7].valid := 1, [2013].log_data[8].valid := 1, [2013].log_data[9].valid := 1, [2013].log_data[10].valid := 1, [2013].log_data[11].valid := 1, [2013].log_data[12].valid := 1, [2013].log_data[13].valid := 1, [2013].log_data[14].valid := 1, [2013].log_data[15].valid := 1, [2013].log_data[16].valid := 1, [2013].log_data[17].valid := 1, [2013].log_data[18].valid := 1, [2013].log_data[19].valid := 1,
